    IF fbStateTimer.Q THEN
      fbStateTimer(IN:=FALSE);
      _nStarts := _nStarts + 1;
      IF bScriptAlive THEN
        nState := cStateRunning;    // is already running
      ELSE  
        RunPythonScript();          // start script
        nState := cStartScript;
			END_IF
		END_IF
  
  //Start Python script and wait until it starts
  cStartScript    :
    fbStateTimer(IN:=TRUE);
    _bBusy := TRUE;

    IF NOT fBScriptLauncher.bBusy AND bScriptAlive THEN 
      IF fBScriptLauncher.bError THEN //Launch error
        LogError(F_Concat2('Script start error=', TO_STRING(fBScriptLauncher.nErrId)));
        nState := cStateError;
      ELSE //Launch done and heartbeat ok
        nState := cStateRunning;
        fbStateTimer(IN:=FALSE);
			END_IF
    ELSIF fbStateTimer.Q THEN //Timeout error (could not start)
      IF fBScriptLauncher.bError THEN //Launch error
        ///LogError(F_Concat2('Script start error=', TO_STRING(fBScriptLauncher.nErrId)));
        LogError(F_Concat2('Script start error=', F_GetAdsErrStr(fBScriptLauncher.nErrId)));
      ELSE
        LogError('Script start error');
      END_IF
      nState := cStateError;
		END_IF
 
  //Script running with correct watchdog feedback
  cStateRunning   : 
    fbStateTimer(IN:=_bJobStartRequest);
    _bBusy := _bJobStartRequest;
    _bJobStopRequest := FALSE;
    _nStarts := 0;
    
    IF _bJobStartRequest AND bPythonNewJobDone THEN
      _bJobStartRequest:=FALSE;
      bPythonNewJobDone := FALSE; 
      fbStateTimer(IN:=FALSE);  
      nState := cStateJobActive;
    ELSIF NOT bScriptAlive THEN //Watchdog error
      LogError('Script watchdog error');
      nState := cStateError;
    ELSIF fbStateTimer.Q THEN //Job timeout error
      LogError('Script new job done error');
      nState := cStateError;
    ELSIF NOT bEnable THEN
      nState := cStateStop;
		END_IF
  
  //JobStarted
  cStateJobActive :
    fbStateTimer(IN:=_bJobStopRequest);
    _bBusy := _bJobStopRequest;
    
    IF _bJobStopRequest THEN
      nPythonNewJob := 0;
    END_IF;  
    
    IF _bJobStopRequest THEN
      _bJobStopRequest:=FALSE;
      fbStateTimer(IN:=FALSE);  
      nState := cStateRunning;
    ELSIF NOT bScriptAlive THEN //Watchdog error
      LogError('Script watchdog error');
      nState := cStateError;
    ELSIF fbStateTimer.Q THEN //Job timeout error
      LogError('Script new job done error');
      nState := cStateError;
    ELSIF NOT bEnable THEN
      nState := cStateStop;
		END_IF
  
  //Error  
  cStateError     :
    fbStateTimer(IN:=FALSE);  
    _bJobStartRequest:=FALSE;
    _bJobStopRequest:=FALSE;
    // reset error 
    IF _bResetError THEN
      _nStarts := 0;          // exit error 
      _nErrCtr := _nErrCtr + 1;
      nState := cStateStop ;
    ELSIF NOT bEnable THEN
      nState := cStateStop ;  // just stop
    ELSIF (_bKeepAlive AND _nStarts <= cMaxStartAttempts)  THEN
      _nErrCtr := _nErrCtr + 1;   // retry 
      nState := cStateStop ;
		END_IF
    
  //Stop 
  cStateStop  :
    StopPythonScript();
    nState := cStateStopping;

  // Stopping
  cStateStopping  :
    IF NOT fBScriptLauncher.bBusy THEN 
      IF fBScriptLauncher.bError THEN //Launch error
        LogError(F_Concat2('Script stop errror:', TO_STRING(fBScriptLauncher.nErrId)));
			END_IF
      nState := cStateIdle;
    END_IF

END_CASE
END_ACTION

METHOD JobStart
VAR_INPUT
  aJobName       : T_MaxString;
  aJobGuid       : T_MaxString;
  nJobImageWidth : UDINT;
  nJobImageHeigth  : UDINT;
  nCamFrameWidth : UDINT;
  pGridSettings  : POINTER TO ST_DefGridSettings;
END_VAR
_bJobStartRequest := TRUE;
_nJobIdCtr := _nJobIdCtr + 1;
nPythonNewJob := _nJobIdCtr;

aPythonJobName := aJobName;
aPythonJobGuid := aJobGuid;
nPythonImageWidth := nJobImageWidth * GVL_Deformation.nC_GridSubReso;
nPythonImageHeight :=nJobImageHeigth * GVL_Deformation.nC_GridSubReso;
nPythonCamFrameWidth := nCamFrameWidth * GVL_Deformation.nC_GridSubReso;
IF pGridSettings <> 0 THEN
  nPythonImageOffsetY := pGridSettings^.nGridImageOffsetY * GVL_Deformation.nC_GridSubReso;
  nPythonGridPitchX := pGridSettings^.nGridPitchX * GVL_Deformation.nC_GridSubReso;
  nPythonGridPitchY := pGridSettings^.nGridPitchY * GVL_Deformation.nC_GridSubReso;
  nPythonGridSizeX := pGridSettings^.nGridSizeX * GVL_Deformation.nC_GridSubReso;
  nPythonGridSizeY := pGridSettings^.nGridSizeY * GVL_Deformation.nC_GridSubReso; 
END_IF
END_METHOD

METHOD JobStop : BOOL
VAR_INPUT
END_VAR
_bJobStopRequest:=TRUE;
END_METHOD

{attribute 'monitoring':='call'}
PROPERTY nErrorId : UDINT
GET
nErrorId := _nErrId;
END_GET
END_PROPERTY

(*
  Register CT to script.
  :return: TRUE if success.
*)
METHOD RegisterCT : BOOL
VAR_INPUT
  nCTIdx  : UDINT;  // ct memory index
END_VAR
IF NOT bScriptAlive THEN RETURN; END_IF  // script not ready, ignore request

nContainerToRegister := UDINT_TO_DINT(nCTIdx);
RegisterCT := TRUE;
END_METHOD

METHOD RemoveCT : BOOL
VAR_INPUT
    nCTID : UDINT;
END_VAR
IF NOT bScriptAlive THEN RETURN; END_IF  // script not ready, ignore request

nContainerToDelete := UDINT_TO_DINT(nCTID);

RemoveCT := TRUE;
END_METHOD

METHOD PRIVATE RunPythonScript : BOOL
VAR_INPUT
END_VAR
VAR
  ams_host : STRING;
  ams_port : UINT;
  cmd : STRING;
END_VAR
// config launcher cmd line for script
//   e.g. fBScriptLauncher.Start('172.17.7.143.1.1 851 PRG_PRINT.fbWorkerDefGrid_Python.fbPythonInterface --sim_mode');

// get parameter dynamically
ams_host := PRG_SYSTEMBASE.sO_AmsNetIdLocalHost;  // localhost
ams_port := TwinCAT_SystemInfoVarList._AppInfo.AdsPort;
cmd := F_Concat5(ams_host,' ',TO_STRING(ams_port),' ',sPythonInterfacePath);
fBScriptLauncher.sStartScriptName := 'start.bat';
fBScriptLauncher.sStopScriptName  := 'stop.bat';
fBScriptLauncher.Start(cmd);
END_METHOD

METHOD PRIVATE StopPythonScript
VAR_INPUT
END_VAR
fBScriptLauncher.Stop(nPID := THIS^.nPythonPID);
END_METHOD

{attribute 'monitoring':='call'}
PROPERTY tWatchdogTime : TIME
GET
tWatchdogTime := fbWatchdog.ET;
END_GET
END_PROPERTY

END_FUNCTION_BLOCK

// ---- POUs/Print/DefGrid/FB_StartPositionDummy.TcPOU
(*
  A start position detection function block dummy.
  A dummy implementation to simulate start triggers at desired positions.
*)
FUNCTION_BLOCK FB_StartPositionDummy EXTENDS FB_BasePrint IMPLEMENTS I_StartPosDetect, I_PrintStatusClient, I_Sim
VAR_INPUT
  bTrigger                    : BOOL;       // manual trigger
  lPosition                   : DINT;       // current position [SubPx]
  fSpeed                      : LREAL;      // current speed [m/s]
  fResolution                 : LREAL;      // current print resolution [dpi*SubPx]
END_VAR

VAR
  // properties
  _bSim               : BOOL;       // simulatio mode active (PROPERTY)
  _bCreateTrigger     : BOOL;       // create new CT trigger (PROPERTY)
  _nStartPosX0        : DINT;       // create position for CT (absolut) [SubPx] (PROPERTY)
  _bAutoTrigger       : BOOL;       // automatic sheet triggers
  
  // config
  iJobDefinition      : CalmarCompPrint.I_JobDefinition;
  
  // local helper
  rfNewCT             : RF_TRIG;    // trigger new ct
  nSheetLength        : DINT;       // sheet length in [SubPx]
  nSheetGap           : DINT;       // sheet gap in [SubPx]
  nSheetEndPosition   : DINT;       // sheet end position [SubPx]
  nNextSheetPosition  : DINT;       // next trigger location
  fSheetPerHour       : LREAL;      // sheets per hour
  fSheetSpeed         : LREAL;      // [m/min] speed meter per minute
  tCheckTrigger       : TON;
  
  tCurrentTimeStamp   : T_DCTIME64; // get current timestamp
  fCurrentTimeStamp   : LREAL;      // current timestamp
  fSensorTimeStamp    : LREAL;      // sensor timestamp
  fDeltaDistance      : LREAL;      // distance that the substrate moved between the detection and the treatment of the information [m]
  
  rfTrig_Sim          : RF_TRIG;
END_VAR

VAR PERSISTENT
  // simulation configuration
  fSheetLength   : LREAL := 0.5;    // [m] sheet length (local or per job given)
  fSheetGap      : LREAL := 0.12;   // [m] gap between two sheets
END_VAR

// checks and fixes
IF iJobDefinition = 0 THEN RETURN; END_IF
IF fSpeed = 0 THEN RETURN; END_IF
IF fSheetLength = 0 THEN fSheetLength := 1; END_IF
IF fResolution = 0 THEN fResolution := 600*32; END_IF
rfTrig_Sim(CLK:=_bSim);
IF    rfTrig_Sim.RT THEN SimEnter(); 
ELSIF rfTrig_Sim.FT THEN SimExit(); END_IF

IF NOT _bSim THEN RETURN; END_IF

// calculations
fSheetSpeed := fSpeed * 60;  // [m/s] -> [m/min]
nSheetGap := F_MeterToSubPixel(fPosMeter := fSheetGap, fResoSubPx := fResolution);  // [m] -> [SubPx]
fSheetPerHour := (60*60)/((fSheetLength+fSheetGap)/fSpeed);
nSheetLength := F_MeterToSubPixel(fPosMeter := fSheetLength, fResoSubPx := fResolution);  // [mm] -> [SubPx]
nNextSheetPosition := _nStartPosX0 + nSheetLength + nSheetGap; 
tCheckTrigger(PT:=TO_TIME(((fSheetLength+fSheetGap)/fSpeed)*1000));

// internal trigger creation
IF (lPosition - nNextSheetPosition) > 0 AND _bAutoTrigger THEN
  bTrigger := TRUE;
  tCheckTrigger(IN:=FALSE);
  tCheckTrigger(IN:=TRUE);
END_IF

// on trigger
rfNewCT(CLK := bTrigger, RT => _bCreateTrigger);
IF _bCreateTrigger THEN   // new ct created
  bTrigger := FALSE;  // reset trigger
  
  (* Calculate the current and sensor time stamp (keep old code not really necessary because we use current timestamp)*)
  tCurrentTimeStamp := F_GetCurDcTaskTime64();
  fCurrentTimeStamp := (ULINT_TO_LREAL(tCurrentTimeStamp )) / 1_000_000.0; (*in ms*)
  fSensorTimeStamp  := fCurrentTimeStamp;
  fDeltaDistance := (fCurrentTimeStamp - fSensorTimeStamp) * 0.001 * fSpeed;  (*Distance that the substrate moved between the detection and the treatment of the information [m]*)
  
  // sheet start and sheet end pos in [SubPx]
  _nStartPosX0     := lPosition - F_MeterToSubPixel(fPosMeter := fDeltaDistance, fResoSubPx := fResolution);
  nSheetEndPosition := _nStartPosX0 + nSheetLength;
END_IF

{attribute 'monitoring' := 'call'}
(*Simulation is enabled set/get*)
PROPERTY bSimEnable : BOOL
GET
bSimEnable := _bSim;
END_GET
SET
_bSim := bSimEnable;
END_SET
END_PROPERTY

(*
  A new container detected.
  NOTE: a pulse only
*)
PROPERTY bStartTrig : BOOL
GET
bStartTrig := _bCreateTrigger;
END_GET
END_PROPERTY

(*
  A valid container detected.
*)
PROPERTY bValid : BOOL
GET
bValid := TRUE;
END_GET
END_PROPERTY

METHOD mJobPause
END_METHOD

METHOD mJobStart
VAR_INPUT
	sJobDef	: CalmarCompPrint.I_JobDefinition;
END_VAR
IF sJobDef = 0 THEN LogError('JobStart: no sJobDef given'); RETURN; END_IF

iJobDefinition := sJobDef;    // current job definition
fSheetLength := iJobDefinition.fSubstrateDepth;
END_METHOD

METHOD mJobStop
VAR_INPUT
	sStatus	: CalmarCompPrint.I_JobStatus;
END_VAR
iJobDefinition := 0;    // delete job definition
END_METHOD

METHOD mProduced
VAR_INPUT
	(* current progress*)
	sProgress	: CalmarCompPrint.I_JobProgress;
END_VAR
; // nothing to do
END_METHOD

(*
  Detected start position X0 (absolute) in [SubPx].
*)
PROPERTY nStartPositionX0 : DINT
GET
nStartPositionX0 := _nStartPosX0;
END_GET
END_PROPERTY

METHOD SimEnter : BOOL
LogInfo('Enter start position creator simulation');
_bSim := TRUE;

_nStartPosX0 := lPosition;
nSheetEndPosition := lPosition;
nNextSheetPosition := lPosition;
END_METHOD

METHOD SimExit : BOOL
LogInfo('Exit start position creator simulation');
_bSim := FALSE;
END_METHOD

END_FUNCTION_BLOCK

// ---- POUs/Print/DefGrid/FB_WorkerDefGrid_Delete.TcPOU
FUNCTION_BLOCK FB_WorkerDefGrid_Delete EXTENDS FB_WorkerDefGrid

METHOD PROTECTED  Attach : BOOL
VAR_INPUT
  iCT              : I_CT;                         (*container at triggered event position*)
END_VAR
IF SUPER^.Attach(iCT:=iCT) THEN

  // directyl release & delete the CT 
  Release(iCT:=_pAttachedCt^);

END_IF
END_METHOD

METHOD   mJobStart
VAR_INPUT
	sJobDef	: CalmarCompPrint.I_JobDefinition;
END_VAR
END_METHOD

METHOD  mJobStop
VAR_INPUT
	sStatus	: CalmarCompPrint.I_JobStatus;
END_VAR
END_METHOD

METHOD Release : BOOL
VAR_INPUT
  iCT              : I_CT;                         (*container at triggered event position*)
END_VAR
IF SUPER^.Release(iCT := iCT) THEN
  
  // it's the last worker so distroy attached CT
  IF _pCTM <> 0 THEN
    LogLvl(Lvl:=E_LogSeverity.Debug, Msg:=F_Concat2('DestroyCT: ', TO_STRING(iCT.pCT^.iId)));
    _pCTM^.DestroyCT(iCT:=iCT);
  END_IF
  
END_IF
END_METHOD

METHOD  work
SUPER^.work();

// release should already be done in attach
IF _pAttachedCt <> 0 THEN
  Release(iCT:=_pAttachedCt^);
END_IF
END_METHOD

END_FUNCTION_BLOCK

// ---- POUs/Print/DefGrid/FB_WorkerDefGrid_Print.TcPOU
FUNCTION_BLOCK FB_WorkerDefGrid_Print EXTENDS FB_WorkerDefGrid IMPLEMENTS I_PrintSubsystem
VAR_INPUT
  nEncoderPos           : DINT;   // Absolute virtual encoder
  bHardwareSync         : BOOL;
  bHardwareHold         : BOOL;
  {warning 'TODO: refactor according WorkerPrintWEU offsets in [m] and worker position without DetectToPrintDist?'}
  fPrintStartOffset     : LREAL;  // Offset from Module reference (configurative PU/PM/PG/PA ADS offset)
  fDetectOffset         : LREAL;  // StartDetect to Modoule reference
  fPrintYOffset         : LREAL;  // Y-Shift in ram memory
  fMasterSpeed          : LREAL;  // Speed [m/s]
  fPUElevation          : LREAL;  // PU distance from substrate [m]
  fPUPlate1_Temperature : LREAL;  // PU Plate1 temperature
  fPUPlate2_Temperature : LREAL;  // PU Plate2 temperature
END_VAR

VAR_OUTPUT
  bPrintActive          : BOOL;   // A print is activated / started
END_VAR

VAR
  // print
  // - references
  _pAdsPg            : POINTER TO FB_ADS_PG;      // pg ads reference (for pa)

  // grid specific
  // - references
  _iParamMediator    : I_ParamMediator;
    
  sDefGridSettings   : ST_DefGridSettings;  
  fCurrentColumnPos  : LREAL; // Currently column position
  fCurrentPreCharge  : LREAL; // Currently to be precharged
  nChargedColumns    : UDINT; // Already charged columns

  fbDropSpeedComp    : FB_DropSpeedComp;  
  bShowDropSpeedSetup: BOOL;

  fbPs               : FB_PS;
  fbPa               : FB_PA;
  fB_PcAdapter       : FB_PC_Adapter;

  _fPrintStartOffset : LREAL;   // internal print start offset (distance Cam -> PG1 + PG Offset + PU offset)
  _fWorkerOffset     : LREAL;   // worker offset from X0 static
  _nPosX0            : DINT;    // X0 for last attached CT (detected postion)
  _nPosXS            : DINT;    // XS for last attached CT (shifted print start position)
  _nPosXDelta        : DINT;    // Shift value X0 -> XS
  _fPosY             : LREAL;   // Y shift for last attached CT
  _fCurrentImgDepth  : LREAL;   // Job: current image length [m]
  _nPosDeltaToPrint  : DINT;    // delta pos in [SbuPx] from attach to print
  _bPaStarted        : BOOL;
  _bPaStartRequested : BOOL;
  fBStartTimeout     : TON;
  rTrigSync          : R_TRIG;
  _bForceDefGridOff  : BOOL;    // force deformation grid stream to ph off (send 0)
  _fPrintUnitWidth   : LREAL;   // print unit width [m]
  // grid settings
  _iPhGrid           : I_Correction_Grid;
  _sPhGridHwCfg      : ST_GridHwCfg;
    
  (*grid limit*)
  _fLimitCorrectionX : LREAL;     // correction limit in y (abs) [px]
  _fLimitCorrectionY : LREAL;     // correction limit in y (abs) [px]
  _bGridWasLimited   : BOOL;      // streamed grid was limited
    
  (*Messaging*)
  _bMsgInitialized   : BOOL;
  fb_MsgQueue        : FB_MSG_QUEUE;                        (*Message queue*)
  fb_MsgHandler      : FB_MSG_HANDLER;                      (*Message handler*)
  sL_MsgConfig       : ST_MSG_CONFIG;                       (*Message config*)
  fb_Msg             : ARRAY [1..iC_NUM_MSG] OF FB_MESSAGE; (*Messages*)
END_VAR

VAR PERSISTENT
  _fColumnsToPrecharge : LREAL := nC_COLUMNS_TO_PRECHARGE;
  _fStartShiftOffset   : LREAL := fC_START_SHIFT_OFFSET;
  _fStartShiftFactor   : LREAL := fC_START_SHIFT_FACTOR;
END_VAR

VAR CONSTANT
  iC_NUM_MSG               : UDINT := 5;
  nC_COLUMNS_TO_PRECHARGE  : LREAL := 2.1;
  fC_GRIDPOINT_STREAM_TIME : LREAL := 0.0025;     // time to stream one point [s]
  fC_START_SHIFT_FACTOR    : LREAL := -0.031;
  fC_START_SHIFT_OFFSET    : LREAL := -0.01;
END_VAR

IF NOT bInitialized THEN RETURN; END_IF

//TODO Add error/warnings
bError := FALSE;
nError := 0;

fbDropSpeedComp(fMasterSpeed:=fMasterSpeed, fDropTravelDistance:=fPUElevation);

//Start offset update
IF _fPrintStartOffset <> (fPrintStartOffset) THEN //Worker position changed
  IF _pAttachedCt = 0 THEN //Update only without attached container
    _fPrintStartOffset :=fPrintStartOffset;
	END_IF
END_IF

//Worker position update
IF _fWorkerPosition <> (_fPrintStartOffset + (_fStartShiftOffset + _fStartShiftFactor * fMasterSpeed)) THEN //Worker position changed (camera settings change)
  setupPosition();
END_IF

(*---- Messaging -----------------------*)
IF _bMsgInitialized THEN
  fb_MsgHandler();
  //fB_Msg[1](bI_Status := dfsdfdsf);
  fb_MsgQueue();
END_IF

PROPERTY aPaState : STRING
GET
aPaState := fbPa.aPaState;
END_GET
END_PROPERTY

METHOD PROTECTED  Attach : BOOL
VAR_INPUT
  iCT              : I_CT;                         (*container at triggered event position*)
END_VAR
Attach:=FALSE;

IF SUPER^.Attach(iCT:=iCT) THEN
  // Additional worker checks
    // - job is valid?
  IF _pAttachedCt^.pJob = 0 OR NOT _bJobActive THEN
    Release(iCT:=iCT);
    RETURN;   // do not print
  
  // CT valid & CT present
  ELSIF NOT _pAttachedCt^.bValid OR NOT _pAttachedCt^.bProductPresent THEN
    Release(iCT:=iCT);
    RETURN;   // do not print
  
  // Ignore start due to hardware hold  
  ELSIF bHardwareHold THEN
    _pNewAttached^.AbortDeformation(sReason:=EC_Print.ecPaAbortHold.Desc, Src:=_pEcSrc^, bHideLog:=TRUE);
    Release(iCT:=iCT);
    RETURN;   // do not print
  
  // - OK attach
  ELSE
    Attach := TRUE;
	END_IF
  
  
  //Prepare print station
  sDefGridSettings := _pAttachedCt^.sDefGridSettings;
  // fix some potential errors
  IF sDefGridSettings.nGridPitchX = 0 THEN sDefGridSettings.nGridPitchX :=1024; LogError(F_concat2('grid not configured, set default nGridPitchX=',TO_STRING(sDefGridSettings.nGridPitchX))); END_IF
  IF sDefGridSettings.nGridPitchY = 0 THEN sDefGridSettings.nGridPitchY :=1024; LogError(F_concat2('grid not configured, set default nGridPitchY=',TO_STRING(sDefGridSettings.nGridPitchY))); END_IF
  
  fbPs.bPrintEnable := iCT.bValid AND iCT.bProductPresent;
  fbPs.setGrid(sGrid:=sDefGridSettings);
  nChargedColumns := 0;

  //Start print, PA should be in READY or DONE
  
  // Set X print position
  _nPosX0 :=    _pAttachedCt^.nPosPrint_X0   {warning 'TODO: please write this in DMAX CreateCT CTM'}
              //- General Shift
              - F_MeterToSubPixel(fbDropSpeedComp.fDropPlacementError, _fPrintResolution*_fSubPxResolution); // - drop compensation*)
  _nPosXDelta := F_MeterToSubPixel(_fPrintStartOffset, _fPrintResolution*_fSubPxResolution); // + PG/PA Shift (additional PG offset 0 for firstLine)
  
  _nPosXS := _nPosX0 + _nPosXDelta;
  fB_PcAdapter.setPrintStartPos(nX0:=_nPosXS);
  
  // Set Y print position
  _fPosY := fPrintYOffset;
  fB_PcAdapter.setPrintYShift(nYShift:=FC_LREAL_TO_DINT(_fPosY));

  // check
  IF _nPosXS < nEncoderPos THEN
    LogWarning(Msg:=F_Concat4('Print start position:', TO_STRING(_nPosXS) ,' < Encoder position:', TO_STRING(nEncoderPos)));
	END_IF
  
  // save current distance to print position
  _nPosDeltaToPrint := _nPosXS - _iCTTracker.getPosAbs();   {warning 'TODO: to test if this matches after the change'}
  checkGridTiming();
  
  IF fbPa.printStart() THEN
    _bPaStarted := FALSE;
    _bPaStartRequested := TRUE;
    Attach:=TRUE;
    LogLvl(Lvl:=E_LogSeverity.Debug, F_Concat2('printStart:', _pAttachedCt^.print(0)));  // print container
    LogLvl(Lvl:=E_LogSeverity.Debug, F_Concat4('> XS:', TO_STRING(_nPosXS), ' = X0:', TO_STRING(_nPosX0)));
    LogLvl(Lvl:=E_LogSeverity.Debug, F_Concat4( 
                                         ' + shStartOffs:', TO_STRING(F_MeterToSubPixel(_fPrintStartOffset,_fPrintResolution*_fSubPxResolution)),
                                         ' - shDropComp:', TO_STRING(F_MeterToSubPixel(fbDropSpeedComp.fDropPlacementError,_fPrintResolution*_fSubPxResolution))
                                         ));
  ELSE  
    LogError(Msg:='PA not ready to start at attach');
    Release(iCT := iCT);
	END_IF
  
ELSE
  // parent attach failed case
END_IF
END_METHOD

PROPERTY bJobActive : BOOL
GET
bJobActive := _bJobActive;
END_GET
END_PROPERTY

PROPERTY bPausePrintCanEx : BOOL
GET
bPausePrintCanEx := FALSE; //Not implemented
END_GET
END_PROPERTY

PROPERTY bPcEnabled : BOOL
GET
bPcEnabled := fB_PcAdapter.bPcEnable;
END_GET
END_PROPERTY

PROPERTY bPrintEnabled : BOOL
GET
bPrintEnabled := _bEnable;
END_GET
END_PROPERTY

PROPERTY bPrinting : BOOL
GET
bPrinting := fbPa.bPrinting;
END_GET
END_PROPERTY

PROPERTY bPrintReady : BOOL
GET
bPrintReady := fbPa.bReady;
END_GET
END_PROPERTY

PROPERTY bQueueEmpty : BOOL
GET
bQueueEmpty := NOT fB_PcAdapter.bJobValid;
END_GET
END_PROPERTY

PROPERTY bStartPrintCanEx : BOOL
GET
bStartPrintCanEx := fbPa.bStartCanEx;
END_GET
END_PROPERTY

PROPERTY bStopPrintCanEx : BOOL
GET
bStopPrintCanEx := fbPa.bStopCanEx;
END_GET
END_PROPERTY

METHOD PRIVATE checkGridTiming : BOOL
VAR
END_VAR
// check for timing problems
IF fMasterSpeed <> 0 THEN

  // - check pre-charge at beginning
  IF _fColumnsToPrecharge * fC_GRIDPOINT_STREAM_TIME * _sPhGridHwCfg.nGridRoiRows >= F_SubPixelToMeter(lPosSubPx:=_nPosDeltaToPrint, fResSubPx:=_fPrintResolution*_fSubPxResolution) / fMasterSpeed  THEN
    LogError('Machine too fast for grid stream (for pre-charge at attach)');
  END_IF
  
 // - check charge time needed per columns vs machine speed and grid-sizeY
 IF fC_GRIDPOINT_STREAM_TIME * _sPhGridHwCfg.nGridRoiRows >= F_SubPixelToMeter(lPosSubPx:=TO_DINT(sDefGridSettings.nGridPitchX), fResSubPx:=_fPrintResolution) / fMasterSpeed THEN
   LogError('Machine too fast for grid stream (time rows per column)');
 END_IF

END_IF
END_METHOD

(*
  Limit correction to boundaries
  :return: TRUE if limited
*)
METHOD PRIVATE correctionLimit : BOOL
VAR_INPUT
  pPoint : POINTER TO ST_DeformationPointAccurate;
END_VAR
VAR
  bLimited : BOOL;
  nExeedX, nExeedY : LREAL;
END_VAR
// limit point correction to boundaries and inform
IF    pPoint^.dx >= _fLimitCorrectionX    THEN nExeedX := pPoint^.dx; pPoint^.dx := _fLimitCorrectionX;    bLimited:=TRUE; 
ELSIF pPoint^.dx <= -1*_fLimitCorrectionX THEN nExeedX := pPoint^.dx; pPoint^.dx := -1*_fLimitCorrectionX; bLimited:=TRUE;
ELSIF pPoint^.dy >= _fLimitCorrectionY    THEN nExeedY := pPoint^.dy; pPoint^.dy := _fLimitCorrectionY;    bLimited:=TRUE;
ELSIF pPoint^.dy <= -1*_fLimitCorrectionY THEN nExeedY := pPoint^.dy; pPoint^.dy := -1*_fLimitCorrectionY; bLimited:=TRUE;
END_IF
IF bLimited THEN 
  LogLvl(Lvl:=E_LogSeverity.Warning, Msg:=F_Concat5( 'Point=',TO_STRING(pPoint^.index),
                                                     F_Concat5(' c:r(',TO_STRING(pPoint^.col),'/',TO_STRING(pPoint^.row), ') '),
                                                     F_Concat4('dx:', TO_STRING(nExeedX), ' dy:', TO_STRING(nExeedY)),
                                                     ' correction exceeded limit')); 
END_IF

_bGridWasLimited := SEL(bLimited, FALSE, TRUE);
correctionLimit := bLimited;
END_METHOD

// current job image length in [m]
PROPERTY fImageLength : LREAL
GET
fImageLength := _fCurrentImgDepth;
END_GET
END_PROPERTY

PROPERTY fMaxPrintSpeed : LREAL
GET
fMaxPrintSpeed := 0;  // TODO: when i_pc_adapter has the info from pc/ph
END_GET
END_PROPERTY

(*
  Max. supported speed [m/s], 0 if not available
*)
{attribute 'monitoring':='call'}
PROPERTY fMaxSpeed : LREAL
GET
VAR
  nSpeedMpMin : DINT;
END_VAR
nSpeedMpMin := SEL(bWorkerEnable AND _pAdsPg <> 0, 0, _pAdsPg^.lMaxPrintSpeed);
fMaxSpeed := TO_LREAL(nSpeedMpMin)/60;
END_GET
END_PROPERTY

{attribute 'monitoring':='call'}
PROPERTY fStartShiftFactor : LREAL
GET
fStartShiftFactor := _fStartShiftFactor;
END_GET
SET
_fStartShiftFactor := fStartShiftFactor;
END_SET
END_PROPERTY

{attribute 'monitoring':='call'}
PROPERTY fStartShiftOffset : LREAL
GET
fStartShiftOffset := _fStartShiftOffset;
END_GET
SET
_fStartShiftOffset := fStartShiftOffset;
END_SET
END_PROPERTY

METHOD PROTECTED gridUpdate : BOOL
VAR_INPUT
  bEnableDeformation : BOOL;      // enable correction update, else correction (0/0) is written
  fPosRelToAttach : LREAL;        // position relative to attach of this worker
END_VAR
VAR
  sPoint : ST_DeformationPointAccurate;
  nRow : UDINT;
  bWasSet : BOOL;
  nAvailPoints : UDINT;
  nConvErr : UDINT;
END_VAR
VAR_INST
  nAvailPoints_mem : UDINT;
END_VAR
//TODO: rewrite this method to look cleaner (less if else)
gridUpdate:=TRUE;

// calculate grid column position
IF sDefGridSettings.nGridPitchX <> 0 THEN
  fCurrentColumnPos := fPosRelToAttach / (sDefGridSettings.nGridPitchX * _fSubPxResolution);   // calc grid column position relative to worker
END_IF

//Check for next correction update 
IF fCurrentColumnPos + _fColumnsToPrecharge > nChargedColumns AND nChargedColumns <= sDefGridSettings.nGridSizeX THEN
  IF bEnableDeformation THEN 
    // sync deformation points
    {warning 'TODO FIX: WHILE'}
    fCurrentPreCharge := fCurrentColumnPos + _fColumnsToPrecharge;
    WHILE FLOOR(fCurrentPreCharge) > nChargedColumns AND nChargedColumns <= sDefGridSettings.nGridSizeX DO
      nAvailPoints := _pAttachedCt^.nAvailableGridPoints;
      IF nAvailPoints >= sDefGridSettings.nGridSizeY * (nChargedColumns+1) THEN // Complete column available?
        nAvailPoints_mem := 0;
        LogLvl(Lvl:=E_LogSeverity.Debug, Msg:=F_Concat2('Charge CG col: ',TO_STRING(nChargedColumns)));
        FOR nRow := 0 TO sDefGridSettings.nGridSizeY - 1 DO
          // get points
          IF _pAttachedCt^.getDeformationPoint(nCol:=nChargedColumns, nRow:=nRow, nSel:=0, sPoint=>sPoint, bWasSet=>bWasSet) THEN
          
            IF NOT bWasSet THEN LogWarning(F_Concat5('Point[c(',TO_STRING(nChargedColumns),')/r(', TO_STRING(nRow),')] was not set')); END_IF  
                      
            // correction limitation
            correctionLimit(pPoint:=ADR(sPoint));
            
            // send point
            IF NOT fbPs.newGridPoint(sPoint:=sPoint) THEN
               LogError(Msg:='stream new point failed');
               gridUpdate:=FALSE;
               RETURN;
            END_IF
          ELSE
            LogError(Msg:='get new grid point failed');
            gridUpdate:=FALSE;
          END_IF
        END_FOR
        
        nChargedColumns := nChargedColumns + 1;
      ELSE
        IF nAvailPoints > nAvailPoints_mem THEN // log once or after every update of new available poinst
          LogError(Msg:='point column expected but not available');
        END_IF
        nAvailPoints_mem := nAvailPoints;
        gridUpdate:=FALSE;
        RETURN;
      END_IF 
    END_WHILE
  ELSE
    // send points with no deformation
      FOR nRow := 0 TO sDefGridSettings.nGridSizeY - 1 DO
        MEMSET(destAddr:=ADR(sPoint), fillByte:=0, n:=SIZEOF(sPoint));
        sPoint.col := TO_DINT(nChargedColumns);
        sPoint.row := TO_DINT(nRow);
        IF NOT fbPs.newGridPoint(sPoint:=sPoint) THEN
           LogError(Msg:='stream new point failed');
           gridUpdate:=FALSE;
           RETURN;
        END_IF
    END_FOR
    nChargedColumns := nChargedColumns + 1;
	END_IF
END_IF
END_METHOD

METHOD InitMsg : BOOL
VAR_INPUT
  pMsgInterface : POINTER TO ST_ADS_MSG_IF;
END_VAR
VAR
  nCtr : UDINT;
END_VAR
IF pMsgInterface = 0 THEN RETURN; END_IF

(*Messaging*)
sL_MsgConfig.bI_Enable       := TRUE;
sL_MsgConfig.pI_FbMsgHandler := ADR(fb_MsgHandler);
fb_MsgHandler.pI_MsgQueue    := ADR(fb_MsgQueue);
fb_MsgQueue.pI_MsgInterface  := pMsgInterface;
fb_MsgQueue.cI_MaxElement    := 6;

(*Messages*)
FOR nCtr := 1 TO iC_NUM_MSG DO
  fb_Msg[nCtr].pI_MsgConfig       := ADR(sL_MsgConfig);
  fb_Msg[nCtr].iI_MsgLocation     := 0;
END_FOR
//fb_Msg[1].iI_MsgNumber       := ;
// ...

_bMsgInitialized := TRUE;
END_METHOD

METHOD InitWorkerPrint : BOOL
VAR_INPUT
  pAdsPg                : POINTER TO FB_ADS_PG;       // pg ads reference (worker prints ads)
  iDefGridParamMediator : I_ParamMediator;
  fPrintUnitWidth       : LREAL;     // print unit width [m]
  fLimitCorrectionX     : LREAL;     // correction limit in y (abs) [px]
  fLimitCorrectionY     : LREAL;     // correction limit in y (abs) [px]
END_VAR
IF NOT bInitialized THEN LogError('Base Worker not initialized! call init() before'); RETURN; END_IF
IF pAdspg = 0 THEN LogError('InitWorkerPrint: invalid parameter proviced'); RETURN; END_IF
IF iDefGridParamMediator = 0 THEN bInitialized := FALSE; LogError('Invalid parameter, no valid param mediator'); RETURN; END_IF

// worker specific init
_pAdsPg := pAdsPg;
_iParamMediator := iDefGridParamMediator;

//Print Aggregate
_fPrintUnitWidth   := fPrintUnitWidth;
_fLimitCorrectionX := ABS(fLimitCorrectionX);
_fLimitCorrectionY := ABS(fLimitCorrectionY);

fbPa.bSyncAfterDone := FALSE;
fbPa.init(iPcAdapter := fB_PcAdapter, iPsInterface := fbPs);
END_METHOD

METHOD   mJobStart
VAR_INPUT
	sJobDef	: CalmarCompPrint.I_JobDefinition;
END_VAR
// Config workers static variables
_fCtSecurityReleasePos := F_MeterToSubPixel(fPosMeter:=(1.5 *sJobDef.fImageDepth) /1000, fResoSubPx:=_fPrintResolution*_fSubPxResolution);

IF NOT bWorkerEnable THEN RETURN; END_IF  // only if enabled

fbPa.jobStart(bEndless:=sJobDef.isEndless());

_bJobActive := TRUE;
_fCurrentImgDepth := sJobDef.fImageDepth/1000;

// grid settings update
IF _iPhGrid <> 0 THEN _sPhGridHwCfg := _iPhGrid.getGridHwCfg(); END_IF
END_METHOD

METHOD  mJobStop
VAR_INPUT
	sStatus	: CalmarCompPrint.I_JobStatus;
END_VAR
fbPa.jobStop();
_bJobActive := FALSE;
END_METHOD

PROPERTY pMsgConfig : POINTER TO ST_MSG_CONFIG
GET
pMsgConfig := ADR(sL_MsgConfig);
END_GET
END_PROPERTY

METHOD registerPc : BOOL
VAR_INPUT
  iNewPC : I_PC;
END_VAR
registerPc := fB_PcAdapter.registerPc(iNewPC := iNewPC);
END_METHOD

METHOD registerPh : BOOL
VAR_INPUT
  iPH : I_PH;
END_VAR
//Attach head to print station
IF iPH <> 0 THEN
  fbPs.registerPh(iNewPh:=iPH);
  _iPhGrid := iPH.iGridCorrection;
END_IF
END_METHOD

METHOD setupPosition
IF _pAttachedCt <> 0 THEN RETURN; END_IF    // Update only without attached container

// WorkerPosition =  PU<-CAM + CAM<-SheetDetect + StartShift calculated (with speed)
fPosition := _fPrintStartOffset + (_fStartShiftOffset + _fStartShiftFactor * fMasterSpeed);
END_METHOD

PROPERTY sPcFlags : CalmarCompPrint.ST_PC_FLAGS
GET
sPcFlags := fB_PcAdapter.sPcFlags;
END_GET
END_PROPERTY

PROPERTY sPcState :  CalmarCompPrint.ST_PG_STATUS
GET
VAR
  sJobStatus : ST_JobProgress;
END_VAR
sPcState.bStartPrintCanEx := fBPa.bStartCanEx;
sPcState.bStartPrintExec  := fBPa.bStartExec;
sPcState.bStopPrintCanEx  := fBPa.bStopCanEx;
sPcState.bStopPrintExec   := fBPa.bStopExec;
sPcState.bPausePrintCanEx := FALSE;       // obsolete ???
sPcState.bPausePrintExec  := FALSE;       // obsolete ???
sPcState.bReady           := fB_PcAdapter.bAllReady OR fB_PcAdapter.bAllDone;
sPcState.bError           := fB_PcAdapter.bError;
sPcState.bPrinting        := fB_PcAdapter.bAllPrinting;
sPcState.bLoad            := fB_PcAdapter.bAllPreparing;
sPcState.bArmed           := fB_PcAdapter.bAllPrinting OR fB_PcAdapter.bAllReady OR fB_PcAdapter.bAllDone OR fB_PcAdapter.bAllPreparing;
sPcState.bEnabled         := bWorkerEnable;
sPcState.bStartStrb       := fBPa.bStartStrb;
sPcState.bPcEnabled       := fB_PcAdapter.bPcEnable;
sPcState.lProductCount    := 0;            // obsolete ???
sPcState.sJobStatus       := sJobStatus;   // obsolete ???
END_GET
END_PROPERTY

METHOD  work
VAR
  bDeformErr : BOOL;
  nDeformStep : E_DeformationStep;
END_VAR
SUPER^.work();

(*Update virtual encoder on all controller boards*)
fB_PcAdapter.setEncoderPos(nEncoderPos);
fB_PcAdapter();

(*Call print aggregate*)
rTrigSync(CLK:=bHardwareSync); 
IF rTrigSync.Q THEN fbPa.sync(); END_IF   // external sync
fbPa.bHold := bHardwareHold;              // external hw hold
fbPa();

fBStartTimeout(IN := _bPaStartRequested,PT := T#60MS);

IF _pAttachedCt <> 0 AND bWorkerEnable THEN // Work only with attached container
  
  // check for generic error
  IF _pAttachedCt^.bValid AND bHardwareHold THEN
    // abort during printing
    _pNewAttached^.AbortDeformation(sReason:=EC_Print.ecPaAbortHold.Desc, Src:=_pEcSrc^, bHideLog:=TRUE);
  END_IF

  // Grid update
  bDeformErr := _pAttachedCt^.getDeformationStatus(eDStep=>nDeformStep);
  {warning 'TODO: re-enable gridUpdate()'}
(*
  IF NOT bDeformErr AND nDeformStep >= E_DeformationStep.gridStarted AND NOT _bForceDefGridOff THEN 
    IF NOT gridUpdate(bEnableDeformation:=TRUE) THEN
      _pAttachedCt^.AbortDeformation(sReason:='WorkerPrint: deformation point update failed', Src:=_pEcSrc^);
    END_IF
  ELSE
    // not started or error already --> erase deformation points
    gridUpdate(bEnableDeformation:=FALSE);
  END_IF  
*)  
  // PA control
  IF _bPaStartRequested THEN
    IF fbPa.bPrinting THEN
      _bPaStarted := TRUE;
      _bPaStartRequested := FALSE;
    ELSIF fBStartTimeout.Q THEN //Stop print at timeout to make ready for next container
      _bPaStarted := FALSE;
      _bPaStartRequested := FALSE;
      fbPa.printStop(bSyncedStop:=FALSE);
      _pNewAttached^.AbortDeformation(sReason:=EC_Print.ecPaStartErr.Desc, Src:=_pEcSrc^, bHideLog:=FALSE);
      Release(_pAttachedCt^);
		END_IF
  ELSIF _bPaStarted THEN
    //Release container when all points have been processed
    IF fbPa.bDone OR fbPa.bStop THEN
      _bPaStarted := FALSE;
      Release(_pAttachedCt^);
    (*ELSIF fbpa.bError THEN
      _pNewAttached^.AbortDeformation(sReason:=EC_Print.ecPaPrintErr.Desc, Src:=_pEcSrc^, bHideLog:=FALSE);
      Release(_pAttachedCt^);*)
    END_IF 
	END_IF
END_IF  

bPrintActive := _bPaStarted;

(*Logging config*)
fbPa.LogLevel := LogLevel;
fB_PcAdapter.LogLevel := LogLevel;
END_METHOD

END_FUNCTION_BLOCK

// ---- POUs/Print/DefGrid/FB_WorkerDefGrid_Python.TcPOU
{attribute 'reflection'} 
FUNCTION_BLOCK FB_WorkerDefGrid_Python EXTENDS FB_WorkerDefGrid IMPLEMENTS I_DeformationHandler
VAR_INPUT
END_VAR
VAR_OUTPUT
END_VAR
VAR
  // interface to py script
  fbPythonInterface : FB_PythonInterface;
  // references
  _iParamMediator : I_ParamMediator;
  
  // local copy of settings
  _bNewJob : BOOL;  // new job was activated
  _CamGridSettings : ST_CameraGridSettings;
  _DefGridSettings : ST_DefGridSettings;
  
  // local copy of job setting
  _aJobName         : T_MaxString;
  _aJobGuid         : T_MaxString;
  _fImageWidthM     : LREAL;          // image width in [m]
  _fImageDepthM     : LREAL;          // image depth in [m]
  

  // messages
  fbMsg_PythonNotRunning : FB_MESSAGE;
END_VAR

VAR CONSTANT
  fC_DEFAULT_WOKER_POSITION : LREAL := 0.01;      // default worker position in [m]
END_VAR

METHOD PROTECTED  Attach : BOOL
VAR_INPUT
  iCT              : I_CT;                         (*container at triggered event position*)
END_VAR
Attach := FALSE;
IF SUPER^.Attach(iCT:=iCT) THEN
  // OK, attached (enabled, was ok to be attached)
  IF _pNewAttached = 0 THEN RETURN; END_IF
  
  // setup check
  IF _iParamMediator = 0 THEN Release(iCT:=iCT); LogError('Invalid param mediator'); RETURN; END_IF
  
  // Additional worker checks
  // - do we have a valid job? used mode?
  IF _CamGridSettings.eCameraMode > E_CameraMode.NoCorrection AND (iCT.pJob = 0 OR NOT _bJobActive) THEN
    _pNewAttached^.AbortDeformation(sReason:='No valid job', Src:=_pEcSrc^, bHideLog:=FALSE);
     Release(iCT:=iCT);
     
  ELSIF _CamGridSettings.eCameraMode > E_CameraMode.NoCorrection THEN
    // OK attach
    // -- only create ct if a deformation is active
    IF CreateDefCt(iCT:=iCT) THEN
        // set state
        _pNewAttached^.StartScript(iDeformationHandler:=THIS^);
        // attached
        Attach := TRUE;
    END_IF
  ELSE
    ; // ignore attach
  END_IF
ELSE
  // parent attach failed
END_IF
END_METHOD

(*
  Create/Release virtual ct in deformation handlers.
  :return: TRUE if success
*)
METHOD PRIVATE CreateDefCt : BOOL;
VAR_INPUT
  iCT : I_CT;
END_VAR
IF iCT = 0 THEN RETURN; END_IF

IF _CamGridSettings.eCameraMode >= E_CameraMode.Live THEN
  IF fbPythonInterface.RegisterCT(iCT.pCT^.nMemIndex) THEN
    CreateDefCt := TRUE;
  ELSE
    _pAttachedCt^.AbortDeformation(sReason:='Could not register to script', Src:=_pEcSrc^, bHideLog:=FALSE);
  END_IF
ELSE
  CreateDefCt := TRUE;
END_IF
END_METHOD

METHOD DeleteCachedCt : BOOL
VAR_INPUT
	iCT	: I_CT;
END_VAR
DeleteDefCt(iCT:=iCT);
END_METHOD

(*
  Delete/Release virtual ct in deformation handlers.
  :return: TRUE if sucess
*)
METHOD DeleteDefCt : BOOL
VAR_INPUT
  iCT : I_CT;
END_VAR
IF iCT = 0 THEN RETURN; END_IF

IF _CamGridSettings.eCameraMode >= E_CameraMode.Live THEN
  IF fbPythonInterface.RemoveCT(iCT.pCT^.nMemIndex) THEN
    DeleteDefCt := TRUE;
  ELSE
    LogError('Could not delete ct in script');
  END_IF
END_IF
END_METHOD

METHOD Init
VAR_INPUT
  pMsgConfig : POINTER TO ST_MSG_CONFIG;         // message config
  fPrintResolution : LREAL := 1;                 // print(head) resolution in [dpi]
  fSubPxResolution : LREAL := 1;                 // SubPixel resolution [SubPx], resolution factor (fI_PrintResolution*fI_SubPxResolution=>Output resolution)
  bParallelCT : BOOL;                            // Support parallel processing of CTs
END_VAR
SUPER^.Init(pMsgConfig:=pMsgConfig, fPrintResolution:=fPrintResolution, fSubPxResolution:=fSubPxResolution, bParallelCT:=bParallelCT);

// Init messages
fbMsg_PythonNotRunning.pI_MsgConfig := _pMsgConfigExt;
fbMsg_PythonNotRunning.iI_MsgLocation := TO_INT(ePr_BLK_PU);
fbMsg_PythonNotRunning.iI_MsgNumber := eC_STAG_DEF_SCRIPT_NOT_RUNNING;
END_METHOD

METHOD InitWorkerPython
VAR_INPUT
  aScriptPath : T_MaxString;                     // path to cmd scripts
  //aAmsLocalHost : T_AmsNetID;                    // Ams netId localhost of the pc to run the script
  iDefGridParamMediator : I_ParamMediator;
END_VAR
IF NOT bInitialized OR _pCTM = 0 THEN LogError('Base Worker not initialized! call init() before'); RETURN; END_IF
IF iDefGridParamMediator = 0 THEN bInitialized := FALSE; LogError('Invalid parameter, no valid param mediator'); RETURN; END_IF

// worker specific init
_iParamMediator := iDefGridParamMediator;

fbPythonInterface.Init(
  sCTManagerPath := _pCTM^.sCTDefGridInstancesPath, 
  sScriptPath:=aScriptPath
);
END_METHOD

METHOD mJobStart
VAR_INPUT
	sJobDef	: CalmarCompPrint.I_JobDefinition;
END_VAR
// checks and fix defaults
IF _iParamMediator = 0 THEN LogError('JobStart: invalid parameter configuration'); RETURN; END_IF
IF _fWorkerPosition = 0 THEN _fWorkerPosition := fC_DEFAULT_WOKER_POSITION; LogError(F_Concat3(_name, ': worker position not set, set default=', TO_STRING(fC_DEFAULT_WOKER_POSITION))); END_IF

// configure
_aJobName := sJobDef.aJobName;
_aJobGuid := sJobDef.aJobId;
_fImageDepthM := sJobDef.fImageDepth/1000;
_fImageWidthM := sJobDef.fImageWidth/1000;

_bNewJob := TRUE;
_bJobActive := TRUE;
END_METHOD

METHOD  mJobStop
VAR_INPUT
	sStatus	: CalmarCompPrint.I_JobStatus;
END_VAR
fbPythonInterface.JobStop();
_bJobActive := FALSE;
END_METHOD

METHOD  work
VAR_INPUT
END_VAR
VAR
  i : UDINT;
  tempCt  : POINTER TO FB_ContainerDefGrid;
  bDeformationDone : BOOL;
  bDeformationError : BOOL;
END_VAR
VAR_INST
  rT_EnablePyIf  : R_TRIG;
END_VAR
SUPER^.work();

IF _iParamMediator = 0 THEN F_Report_Error(ErrType:=EN_REPORT_ERROR_TYPE.Report_Error_0Pointer); RETURN; END_IF
_CamGridSettings := _iParamMediator.sCameraGridSettings;
_DefGridSettings := _iParamMediator.sDeformationGridSettings;

// reconfig script after job started (Mediator parameter are defined in JobStart())
IF _bNewJob OR rT_EnablePyIf.Q THEN   // new job activated or re-enabled
  _bNewJob := FALSE;
  
  // setup script
  fbPythonInterface.JobStart(
    aJobName:=_aJobName,
    aJobGuid:=_aJobGuid,
    nJobImageWidth:=DINT_TO_UDINT(F_MeterToSubPixel(fPosMeter:=_fImageDepthM, fResoSubPx:=_fPrintResolution)),
    nJobImageHeigth:=DINT_TO_UDINT(F_MeterToSubPixel(fPosMeter:=_fImageWidthM, fResoSubPx:=_fPrintResolution)),
    nCamFrameWidth:=DINT_TO_UDINT(FC_LREAL_TO_DINT(_CamGridSettings.fGridFeaturePitch)),
    pGridSettings:=ADR(_DefGridSettings)
  );
END_IF

// start/stop script
IF _CamGridSettings.eCameraMode >= E_CameraMode.Live AND THIS^.bWorkerEnable THEN 
  fbPythonInterface.bEnable := TRUE;
ELSE
  fbPythonInterface.bEnable := FALSE;
END_IF
rT_EnablePyIf(CLK:=fbPythonInterface.bEnable);

fbPythonInterface();

IF _pAttachedCt <> 0 THEN
  // nothing to do anymore just release CT
  // NOTE: the delete of the CT is done by DeleteDefCt() method directly into fbPythonInterface
  Release(_pAttachedCt^);
END_IF

// messages
fbMsg_PythonNotRunning(bI_Status:=fbPythonInterface.bError);
IF fbMsg_PythonNotRunning.bMsgAck THEN fbPythonInterface.ackError(); END_IF
END_METHOD

END_FUNCTION_BLOCK

// ---- POUs/Print/DefGrid/FB_WorkerDefGrid_Verify.TcPOU
FUNCTION_BLOCK FB_WorkerDefGrid_Verify EXTENDS FB_WorkerDefGrid
VAR_OUTPUT
  bWateGateActive   AT%Q* : BOOL;     //  wate gate activation pulse
END_VAR
VAR
  bLastEject   : BOOL;   // stores state if last CT TRUE:=Eject, FALSE:=OK
  tpEjectPulse  : TP := (PT:=T#80MS);
  
  // print manager reference
  _pPm : POINTER TO FB_ProdManager_DMAX;
  
  // view verify history
  tpShowResult : TP := (PT:=T#700MS);
  nStateHistory : ARRAY[1..20] OF UINT;   // 2=???, 1=Eject, 0=OK
  nStateHistory_FillColor : ARRAY[1..20] OF UDINT;
  sResultText : STRING;
  
  // Grid Table export
  nCTId : DINT;
  bEnableGridExport : BOOL;
  nExportWrites : UDINT;
  sOutputPath : T_MaxString := 'C:\GridExport';
  sFileFormat : STRING := 'json';
  fbGridExporter : FB_GridDataExporter;
END_VAR

METHOD PROTECTED  Attach : BOOL
VAR_INPUT
  iCT              : I_CT;                         (*container at triggered event position*)
END_VAR
VAR 
  bSuccess         : BOOL;
END_VAR
IF SUPER^.Attach(iCT:=iCT) THEN
  
  // do CT supervision here and decice what happens with this sheet
   bSuccess := TRUE;
  IF NOT iCT.bValid AND iCT.bProductPresent AND iCT.pJob <> 0 THEN
    bSuccess := FALSE;
    // tag for ejection
    iCT.pCT^.lPrOutput := EN_PrinterOutput.trash;
	END_IF

  // finish CT in production
  IF _pPm <> 0 THEN 
    _pPm^.CT_Finish(sCT:=iCT, bSuccess:=bSuccess);      // report to job status
  ELSE
    LogError('PrintManager not set');
	END_IF
  
  // select output
  IF iCT.pCT^.lPrOutput = EN_PrinterOutput.trash THEN
    // create eject trigger
    tpEjectPulse(IN:=TRUE);
    bLastEject := TRUE;
    LogLvl(Lvl:=E_LogSeverity.Debug, Msg:=F_Concat2('Eject CT: ', _pAttachedCt^.print(0)));
  ELSE
    tpEjectPulse(IN:=FALSE);
    bLastEject := FALSE;
	END_IF
  
  // History view
  MEMMOVE(destAddr:=ADR(nStateHistory[1+1]),           srcAddr:=ADR(nStateHistory[1]),           n:=((SIZEOF(nStateHistory)/SIZEOF(nStateHistory[1]))-1)*SIZEOF(nStateHistory[1]));
  MEMMOVE(destAddr:=ADR(nStateHistory_FillColor[1+1]), srcAddr:=ADR(nStateHistory_FillColor[1]), n:=((SIZEOF(nStateHistory_FillColor)/SIZEOF(nStateHistory_FillColor[1]))-1)*SIZEOF(nStateHistory_FillColor[1]));
  
  nStateHistory[1] := SEL(bLastEject=TRUE, 0, 1);
  sResultText := SEL(bLastEject=TRUE, 'OK', 'NOK');

  IF iCT.bProductPresent AND iCT.bValid THEN        nStateHistory_FillColor[1] := 16#FF000000 OR WebColors.LightGreen.lCode;
  ELSIF iCT.bProductPresent AND NOT iCT.bValid AND iCT.pCT^.lPrOutput = EN_PrinterOutput.trash THEN nStateHistory_FillColor[1] := 16#FF000000 OR WebColors.LightSalmon.lCode;   
  ELSIF iCT.bProductPresent AND NOT iCT.bValid AND iCT.pCT^.lPrOutput <> EN_PrinterOutput.trash THEN nStateHistory_FillColor[1] := 16#FF000000 OR WebColors.LightGray.lCode;
	ELSIF NOT iCT.bProductPresent THEN                nStateHistory_FillColor[1] := 16#FF000000 OR WebColors.LightGray.lCode;
  END_IF

  tpShowResult(IN:=FALSE);
  tpShowResult(IN:=TRUE);
  
  // grid history
  IF bEnableGridExport AND iCT.bProductPresent AND nExportWrites < 100 THEN
    nCTId := _pAttachedCt^.pCT^.iId;
    sFileFormat := SEL(sFileFormat='csv', 'json', 'csv');
    fbGridExporter(
        sOutputDir:=sOutputPath,
        sFileName:=F_Concat4('\Export_', TO_STRING(nCTId), '.', sFileFormat),
        pFbImageDeformation:=_pAttachedCt^.pImageDeformation,
        //nSelectGrid:=
    );
    fbGridExporter.startExport();
    nExportWrites:=nExportWrites+1;
  ELSE
    nExportWrites := 0; bEnableGridExport := FALSE;
  END_IF
END_IF
END_METHOD

(*
  Set PrintManager.
*)
METHOD InitWorkerVerify : BOOL
VAR_INPUT
  pPm : POINTER TO FB_ProdManager_DMAX;
END_VAR
IF pPm = 0 THEN LogError('Invalid Pm given'); END_IF

_pPm := pPm;  // register print manager reference
END_METHOD

METHOD   mJobStart
VAR_INPUT
	sJobDef	: CalmarCompPrint.I_JobDefinition;
END_VAR
END_METHOD

METHOD  mJobStop
VAR_INPUT
	sStatus	: CalmarCompPrint.I_JobStatus;
END_VAR
END_METHOD

METHOD Release : BOOL
VAR_INPUT
  iCT              : I_CT;                         (*container at triggered event position*)
END_VAR
IF SUPER^.Release(iCT := iCT) THEN
  ;
END_IF
END_METHOD

METHOD  work
VAR_INST
  fT_Pulse  : F_TRIG;
END_VAR
SUPER^.work();

// output signal handling
tpEjectPulse(Q=>bWateGateActive);
fT_Pulse(CLK:=bWateGateActive);
tpShowResult();
//IF tpShowResult.IN:=TRUE AND NOT tpShowResult.Q THEN tpShowResult(IN:=FALSE); END_IF   // reset pulse

fbGridExporter();

// release
IF tpEjectPulse.IN THEN
  IF fT_Pulse.Q THEN  
    tpEjectPulse(IN:=FALSE);
  END_IF
END_IF

IF _pAttachedCt <> 0 THEN   // just release any attached container in this cycle
  Release(iCT:=_pAttachedCt^);
END_IF
END_METHOD

END_FUNCTION_BLOCK

// ---- POUs/Print/FB_SheetDetectSupervision.TcPOU
FUNCTION_BLOCK FB_SheetDetectSupervision
VAR_INPUT
  IbSensorSheetCalender                   AT%I* : BOOL;            // Sensor signal B250
  IbSensorSheetInlet                      AT%I* : BOOL;            // Sensor signal B257
  IbSensorSheetOutlet                     AT%I* : BOOL;            // Sensor signal B254

  InCurrentPos                                  : DINT;            // Current position in [SubPx]
  IbMachineStopped                              : BOOL;            // Machine stopped
  IbInhibitSheetTrigger                         : BOOL;            // inhibit trigger signals for substrate length
  IbCameraTrigger                               : BOOL;            // Camera trigger
END_VAR

VAR_OUTPUT
  ObSheetJamPrintingSystem                AT%Q* : BOOL;            // Sheet jam in printing system detected

  ObCameraTriggerEnable                         : BOOL;            // Camera trigger enable
  ObCameraTriggerIncorrect                      : BOOL;            // Camera trigger incorrect
  ObCameraTriggerSupervison                     : BOOL;            // Camera trigger supervision for sheet jam
  ObSheetDetectFree                             : BOOL;            // sheet detect sensors are free
END_VAR

VAR
  _PrintSubPixelResolution                      : UDINT := 600 * 32;           // Print sub pixel resolution

  fbSheetDetectRingbuffer01                     : FB_RINGBUFFER;
  fbSheetDetectRingbuffer02                     : FB_RINGBUFFER;

  rfTrig_CameraTriggerSupervison                : RF_TRIG;
  bCameraTriggerSupervisonOn                    : BOOL;
  
  rfTrig_MachineStopped                         : RF_TRIG;

  // jam event
  rTrig_SheetJam                                : R_TRIG;
  _bSheetJamEvent                               : BOOL;
  
  // error handling 
  nConversionErrorCounter                       : UDINT;
END_VAR

VAR PERSISTENT
  RemSheetDetectSupervisionPar                  : ST_SheetDetectSupervisionPar;
END_VAR

rfTrig_MachineStopped(CLK := IbMachineStopped);

(*B250 => B256*)
fbSheetDetectRingbuffer01.pI_ConversionErr      := ADR(nConversionErrorCounter);
fbSheetDetectRingbuffer01.bI_Reset              := IbMachineStopped;
fbSheetDetectRingbuffer01.bI_Sensor             := NOT IbSensorSheetCalender;
fbSheetDetectRingbuffer01.iI_CurrentPos         := DINT_TO_UDINT(InCurrentPos);
fbSheetDetectRingbuffer01.iI_Pg_Offset          := 0;
fbSheetDetectRingbuffer01.iI_Offset_X0          := fbSheetDetectRingbuffer01.iI_CurrentPos + DINT_TO_UDINT(F_MeterToSubPixel(RemSheetDetectSupervisionPar.fR_SheetDetectDistance01, UDINT_TO_LREAL(_PrintSubPixelResolution)));           
fbSheetDetectRingbuffer01.iI_Resolution         := UDINT_TO_INT(_PrintSubPixelResolution);
fbSheetDetectRingbuffer01.fI_ShiftDistance      := 0 - RemSheetDetectSupervisionPar.fR_SheetDetectRange01_m;
fbSheetDetectRingbuffer01();

(*B256 => B254*)
fbSheetDetectRingbuffer02.pI_ConversionErr      := ADR(nConversionErrorCounter);
fbSheetDetectRingbuffer02.bI_Reset              := IbMachineStopped;
fbSheetDetectRingbuffer02.bI_Sensor             := IbCameraTrigger;
fbSheetDetectRingbuffer02.iI_CurrentPos         := DINT_TO_UDINT(InCurrentPos);
fbSheetDetectRingbuffer02.iI_Pg_Offset          := 0;
fbSheetDetectRingbuffer02.iI_Offset_X0          := fbSheetDetectRingbuffer02.iI_CurrentPos + DINT_TO_UDINT(F_MeterToSubPixel(RemSheetDetectSupervisionPar.fR_SheetDetectDistance02, UDINT_TO_LREAL(_PrintSubPixelResolution)));           
fbSheetDetectRingbuffer02.iI_Resolution         := UDINT_TO_INT(_PrintSubPixelResolution);
fbSheetDetectRingbuffer02.fI_ShiftDistance      := 0 - RemSheetDetectSupervisionPar.fR_SheetDetectRange02_m;
fbSheetDetectRingbuffer02();

RemSheetDetectSupervisionPar.nR_SheetDetectRange01_SubPx := F_MeterToSubPixel(REAL_TO_LREAL(RemSheetDetectSupervisionPar.fR_SheetDetectRange01_m), UDINT_TO_LREAL(_PrintSubPixelResolution));
RemSheetDetectSupervisionPar.nR_SheetDetectRange02_SubPx := F_MeterToSubPixel(REAL_TO_LREAL(RemSheetDetectSupervisionPar.fR_SheetDetectRange02_m), UDINT_TO_LREAL(_PrintSubPixelResolution));

IF RemSheetDetectSupervisionPar.bR_Enable THEN
  (*Masking sheet detection of camera system*)
  ObCameraTriggerEnable     :=     (InCurrentPos > (fbSheetDetectRingbuffer01.iO_ShiftOffset_X0 - RemSheetDetectSupervisionPar.nR_SheetDetectRange01_SubPx)) 
                               AND (InCurrentPos < (fbSheetDetectRingbuffer01.iO_ShiftOffset_X0 + RemSheetDetectSupervisionPar.nR_SheetDetectRange01_SubPx));
  (*Sheet trigger was incorrect because of faulty detection*)
  IF NOT ObCameraTriggerEnable AND IbSensorSheetInlet AND NOT IbInhibitSheetTrigger THEN
    ObCameraTriggerIncorrect := TRUE;
  END_IF

  (*Sheet jam supervision*)
  ObCameraTriggerSupervison :=     (InCurrentPos > (fbSheetDetectRingbuffer02.iO_ShiftOffset_X0 - RemSheetDetectSupervisionPar.nR_SheetDetectRange02_SubPx)) 
                               AND (InCurrentPos < (fbSheetDetectRingbuffer02.iO_ShiftOffset_X0 + RemSheetDetectSupervisionPar.nR_SheetDetectRange02_SubPx));
  rfTrig_CameraTriggerSupervison(CLK := ObCameraTriggerSupervison);
  IF rfTrig_CameraTriggerSupervison.RT THEN
    bCameraTriggerSupervisonOn := TRUE;
  END_IF
  IF bCameraTriggerSupervisonOn AND IbSensorSheetOutlet THEN
    bCameraTriggerSupervisonOn := FALSE;
  END_IF
  IF rfTrig_CameraTriggerSupervison.FT AND bCameraTriggerSupervisonOn THEN
    ObSheetJamPrintingSystem   := TRUE;
    bCameraTriggerSupervisonOn := FALSE;
  END_IF

  ObSheetDetectFree := TRUE;
  IF IbMachineStopped THEN
    ObCameraTriggerIncorrect   := FALSE;
    bCameraTriggerSupervisonOn := FALSE;

    IF NOT IbSensorSheetCalender OR IbSensorSheetInlet OR IbSensorSheetOutlet THEN
      ObSheetDetectFree := FALSE;
    END_IF
  END_IF
  IF rfTrig_MachineStopped.FT THEN
    ObSheetJamPrintingSystem   := FALSE;
  END_IF
ELSE
  ObCameraTriggerEnable     := TRUE;
  ObCameraTriggerIncorrect  := FALSE;
  ObSheetJamPrintingSystem  := FALSE;
  ObSheetDetectFree         := TRUE;
END_IF

rTrig_SheetJam(CLK:=ObSheetJamPrintingSystem);
IF rTrig_SheetJam.Q THEN _bSheetJamEvent := TRUE; END_IF

PROPERTY bSheetJamEvent : BOOL
GET
bSheetJamEvent := _bSheetJamEvent;
_bSheetJamEvent := FALSE;
END_GET
END_PROPERTY

PROPERTY PrintSubPixelResolution : UDINT
SET
_PrintSubPixelResolution := PrintSubPixelResolution;
END_SET
END_PROPERTY

END_FUNCTION_BLOCK

// ---- GlobalTextList.TcGTLO
TEXTLIST GlobalTextList
  10210 = '  x:%0.5f'
  6570 = '  y:%0.5f'
  781 = ' Camera offset Y [mm]: %f'
  2961 = ' cM: Camera start margin [m]: %f'
  5665 = ' Modus: %s'
  13668 = ' Nb teach marks: %d'
  13672 = ' Nb teach sectors: %d'
  9596 = ' Number of marks: %d'
  10437 = ' pW: Actual PrintUnit width [m]: %f'
  8296 = ' pWc: PrintUnit width [m]: %f'
  2948 = ' Sector of transmission: %d'
  5660 = ' Version number: %d'
  1184 = '%0.01f'
  14098 = '%0.02f'
  4085 = '%0.02f m/s'
  13676 = '%0.04f'
  8040 = '%0.06f'
  303 = '%0.0f'
  2502 = '%0.0f [m]'
  8178 = '%0.0f [px]'
  293 = '%0.1f'
  11885 = '%0.1f [cols]'
  430 = '%0.1f [m/min]'
  941 = '%0.1f [um]'
  10 = '%0.2f'
  993 = '%0.3f'
  1945 = '%0.3f [m/min]'
  6769 = '%0.3f [m/s]'
  4949 = '%0.3f [ms]'
  10891 = '%0.3f [m]'
  7216 = '%0.3f [px]'
  1864 = '%0.4f'
  11719 = '%0.4f  [m]'
  1796 = '%0.4f [ms]'
  7315 = '%0.4f [m]'
  1072 = '%0.5f'
  1822 = '%0.5f [m]'
  1887 = '%0.6f [m/s]'
  1147 = '%0.6f [ms]'
  820 = '%0.6f [m]'
  2289 = '%0.6f [um]'
  704 = '%1.1f'
  3079 = '%1.1f mm'
  3009 = '%1.1f mm/s'
  1930 = '%1.2f'
  741 = '%1.2f mm'
  3014 = '%1.3f mm'
  2489 = '%1.3f [mm]'
  6533 = '%1.3f [px]'
  3085 = '%1.4f m'
  7362 = '%1.4f [ms]'
  2560 = '%1.4f [m]'
  3481 = '%1.5f [m]'
  9 = '%d'
  3602 = '%d [px]'
  2955 = '%d [um]'
  456 = '%f'
  2383 = '%f [m/min]'
  5388 = '%f [mm]'
  812 = '%f [m]'
  2912 = '%f [s.p.min]'
  3959 = '%f [um]'
  27 = '%s'
  260 = '%s%%'
  9843 = '(Hw)Enable'
  3930 = '(not used) CameraToPrintUnit'
  17381 = '(viratual) generated'
  12232 = '*'
  447 = '+'
  7024 = '+/- %0.4f'
  8411 = '-'
  68 = '/'
  2589 = '1'
  2552 = '1. Activate (Drop)SpeedComp with Time set to 0\n\n2. Test print with production speed1\n   -> Measure displacement with Speed1\n\n3. Test print with production speed2\n   -> Measure displacement with Speed2\n\n4. Enter Speed and Displacement values in\n    table for Test1 and Test2\n\n5. Start new Time calculation'
  245 = '1. Activate (Drop)SpeedComp with Time set to 0\n\n2. Test print with Speed1\n   -> Measure displacement with Speed1\n\n3. Test print with Speed2\n   -> Measure displacement with Speed2\n\n4. Enter Speed and Displacement values in\n    table for Test1 and Test2\n\n5. Start new Time calculation'
  864 = '1. Activate (Drop)SpeedComp with Time set to 0\n\n2. Test1 print with production speed1\n   -> Measure displacement with Speed1\n\n3. Test2 print with production speed2\n   -> Measure displacement with Speed2\n\n4. Enter Speed and Displacement values in\n    table for Test1 and Test2\n\n5. Start new Time calculation'
  835 = '1. Activate (Drop)SpeedComp with Time set to 0\n\n2. Test1: print with production speed1\n   -> Measure displacement with Speed1\n\n3. Test2: print with production speed2\n   -> Measure displacement with Speed2\n\n4. Enter Speed and Displacement values in\n    table for Test1 and Test2\n\n5. Start new Time calculation'
  41 = '1. Activate DropSpeeCmp'
  1428 = '1. Activate DropSpeeComp\n   + Set Time to 0'
  1322 = '1. Activate DropSpeeComp\n   + Set Time to 0\n\n\n\n'
  1646 = '1. Activate DropSpeeComp\n   + Set Time to 0\n\n2. Test print with Speed1\n   + Measure displacement with Speed1\n\n'
  478 = '1. Activate DropSpeeComp\n   + Set Time to 0\n\n2. Test print with Speed1\n   + Measure displacement with Speed1\n\n3. Test print with Speed2\n   + Measure displacement with Speed2\n'
  2206 = '1. Activate DropSpeeComp\n   + Set Time to 0\n\n2. Test print with Speed1\n   + Measure displacement with Speed1\n\n3. Test print with Speed2\n   + Measure displacement with Speed2\n\n\n4. Enter values in table for Test1 and Test2\n\n5. Start new Time calculation'
  543 = '1. Activate DropSpeeComp\n   + Set Time to 0\n\n2. Test print with Speed1\n   + Measure displacement with Speed1\n\n3. Test print with Speed2\n   + Measure displacement with Speed2\n\n\n\n4. Enter values in table for Test1 and Test2'
  1417 = '1. Activate DropSpeeComp\n   + Set Time to 0\n\n2. Test print with Speed1\n   + Measure displacement with Speed1\n\n3. Test print with Speed2\n   + Measure displacement with Speed2\n\n5. Start new Time calculation\n\n4. Enter values in table for Test1 and Test2'
  2118 = '1. Activate DropSpeeComp\n   Set Time to 0'
  1160 = '1. Activate DropSpeeComp with Time set to 0\n\n2. Test print with Speed1\n   + Measure displacement with Speed1\n\n3. Test print with Speed2\n   + Measure displacement with Speed2\n\n\n4. Enter values in table for Test1 and Test2\n\n5. Start new Time calculation'
  1763 = '1. Activate DropSpeeComp with Time set to 0\n\n2. Test print with Speed1\n   + Measure displacement with Speed1\n\n3. Test print with Speed2\n   + Measure displacement with Speed2\n\n4. Enter values in table for Test1 and Test2\n\n5. Start new Time calculation'
  1928 = '1. Activate DropSpeeComp with Time set to 0\n\n2. Test print with Speed1\n   -> Measure displacement with Speed1\n\n3. Test print with Speed2\n   -> Measure displacement with Speed2\n\n4. Enter Speed and Displacement values\n     in table for Test1 and Test2\n\n5. Start new Time calculation'
  2230 = '1. Activate DropSpeeComp with Time set to 0\n\n2. Test print with Speed1\n   -> Measure displacement with Speed1\n\n3. Test print with Speed2\n   -> Measure displacement with Speed2\n\n4. Enter Speed and Displacement values in\n    table for Test1 and Test2\n\n5. Start new Time calculation'
  2617 = '1. Activate DropSpeeComp with Time set to 0\n\n2. Test print with Speed1\n   -> Measure displacement with Speed1\n\n3. Test print with Speed2\n   -> Measure displacement with Speed2\n\n4. Enter Speed and Displacement values in     table for Test1 and Test2\n\n5. Start new Time calculation'
  167 = '1. Activate DropSpeeComp with Time set to 0\n\n2. Test print with Speed1\n   -> Measure displacement with Speed1\n\n3. Test print with Speed2\n   -> Measure displacement with Speed2\n\n4. Enter Speed and Displacement values in table for Test1 and Test2\n\n5. Start new Time calculation'
  1944 = '1. Activate DropSpeeComp with Time set to 0\n\n2. Test print with Speed1\n   -> Measure displacement with Speed1\n\n3. Test print with Speed2\n   -> Measure displacement with Speed2\n\n4. Enter values in table for Test1 and Test2\n\n5. Start new Time calculation'
  363 = '1. Activate DropSpeedComp with Time set to 0\n\n2. Test print with Speed1\n   -> Measure displacement with Speed1\n\n3. Test print with Speed2\n   -> Measure displacement with Speed2\n\n4. Enter Speed and Displacement values in\n    table for Test1 and Test2\n\n5. Start new Time calculation'
  2048 = '1. Active DropSpeedComp'
  2104 = '1. Set Time to 0'
  7016 = '2*a'
  1505 = '2. Test print with Speed1\n   + Measure displacement with Speed1'
  2308 = '2. Test print with Speed1\n   Measure displacement with Speed1'
  1658 = '3. Test print with Speed2\n   + Measure displacement with Speed2'
  77 = '3. Test print with Speed2\n   Measure displacement with Speed2'
  550 = '4. Calculate new Time'
  581 = '4. Enter values in table for Test1 and Test2'
  1286 = '4. Start new Time calculation'
  2168 = '4p PLC'
  739 = '5. Start new Time calculation'
  8190 = '<'
  11083 = '<-'
  448 = '='
  6003 = '>'
  9654 = '>Camera(s)'
  1163 = '>FineAlignement'
  15769 = '>PrintPosition'
  18969 = '>WorkerPrint PG1 (Row1)'
  2212 = '>WorkerPrint PG2 (Row2)'
  19156 = 'a'
  14960 = 'a (mark size)'
  3758 = 'a/2'
  7335 = 'a: %d'
  4185 = 'Abort'
  3571 = 'Acknowledge'
  1383 = 'Act pos.'
  140 = 'Active'
  1300 = 'active camera device'
  517 = 'active camera device type'
  7324 = 'active camera mode'
  2160 = 'Actual Y-Resolution [dpi]: %1.4f'
  8699 = 'added points'
  1427 = 'ADS axis position'
  590 = 'ADS Axis Position'
  5009 = 'ADS command'
  717 = 'ADS Commands'
  9674 = 'ADS PG shift'
  2259 = 'ADS PU shift'
  4169 = 'ADS settings'
  723 = 'ADS Settings'
  15944 = 'All Epsitron'
  3353 = 'All Epsitron OK'
  5267 = 'All Inputs ok'
  5680 = 'AnalogMaxDigit'
  3775 = 'Auto'
  671 = 'AUTO/MANU CONTROL'
  4177 = 'Automatic Mode'
  1339 = 'Automatic or ManualTeach'
  2606 = 'AutomaticMode or ManualTeach'
  12039 = 'b'
  7246 = 'b (mark size)'
  9731 = 'B250'
  2262 = 'B254'
  16217 = 'B257'
  2111 = 'Back'
  608 = 'Bacl'
  3856 = 'bStopReady'
  210 = 'Busy'
  19400 = 'by calculation'
  6619 = 'C'
  411 = 'c'
  9048 = 'c (mark distance)'
  744 = 'C1'
  743 = 'C2'
  1065 = 'c: %d'
  3129 = 'c:%d'
  710 = 'Ca/Pu'
  136 = 'Calculate new time'
  1431 = 'Calculate new Time'
  13216 = 'Calender'
  6811 = 'cam simulation'
  1299 = 'Cam valid'
  1186 = 'Cam Valid'
  4259 = 'Camera'
  13991 = 'Camera activated'
  11573 = 'Camera Detail: %s'
  1141 = 'Camera ip address'
  1321 = 'camera mode desired'
  530 = 'camera mode desired (active cam)'
  1086 = 'Camera name'
  1061 = 'camera port'
  2103 = 'Camera sink'
  6170 = 'Camera temperature [°C]: %1.1f'
  5051 = 'Camera trigger'
  1990 = 'Camera type'
  9680 = 'Camera->PU'
  11139 = 'CameraToPrintUnit'
  8862 = 'CameraTrigger'
  14480 = 'CamPointsFifo'
  5607 = 'CamToPU'
  5019 = 'CanEx'
  7354 = 'cfb'
  10808 = 'Charged columns'
  8294 = 'Check delay'
  708 = 'Clean'
  3790 = 'Clean Active'
  719 = 'Clean after Capping'
  720 = 'Clean after Purge'
  1935 = 'Clean Head'
  1246 = 'Clean head (max %d)'
  711 = 'Clean Unit'
  15882 = 'Clean unit (max %d)'
  14428 = 'CleanCappPosition'
  4247 = 'CLEANER'
  4468 = 'Cleaner pump'
  265 = 'Cleaning'
  3760 = 'Cleaning Operations'
  740 = 'Cleaning Safe '
  4828 = 'CleaningProcess'
  212 = 'col'
  1396 = 'Column Precharge'
  6407 = 'Comp.'
  10565 = 'Compensation temperatur extension'
  11736 = 'configured camera mode, active=%s'
  10779 = 'Connected'
  9558 = 'constant'
  7336 = 'correction relative'
  6221 = 'csv'
  8478 = 'ct'
  3579 = 'CT'
  8221 = 'CT @Deformation (more corrections followed @Print!)'
  1165 = 'CT Id=%d'
  5554 = 'CT ImageDeformation'
  1850 = 'CT PrintRef'
  6824 = 'CT Status'
  17584 = 'CTDetail  @PrintWorker[1]  !No FineAlignment yet applied!'
  11030 = 'CTManager'
  15305 = 'Current'
  69 = 'current camera mode (active cam)'
  1219 = 'Current columen relative to Worker Attach'
  6060 = 'Current column'
  10240 = 'Current CT'
  10438 = 'Current position'
  10758 = 'Current reso used (from machine)'
  20158 = 'Current Speed'
  4981 = 'Current step'
  1573 = 'CurrentSpeed [m/s]'
  389 = 'D'
  2060 = 'Dead Time'
  1132 = 'Dead/Add Time'
  4013 = 'Dead/Add Time [ms]'
  21105 = 'Debug & Simulation'
  12899 = 'Deformation'
  1100 = 'DeformType'
  3003 = 'Delta P'
  2040 = 'Detect -> Cam'
  7545 = 'Detect -> Cam (Trig.Dist.)'
  18521 = 'Detected'
  6 = 'detected length [mm]'
  10000 = 'detected length [m]'
  1172 = 'Detected Marks: %d'
  9097 = 'Detection'
  10216 = 'Detection range [m]'
  12392 = 'DetectToCam'
  11747 = 'DetectToCamera'
  1597 = 'Device type'
  4990 = 'DevOpActive'
  5555 = 'Diff [mm]'
  8247 = 'Diff [m]'
  16644 = 'Direction'
  1171 = 'Disable left SLM'
  6432 = 'Disable right SLM'
  2162 = 'Displacement'
  1297 = 'Displacment'
  4696 = 'Distance in [p]'
  16193 = 'Distance [m]'
  4984 = 'DistBetweenMasks'
  3424 = 'DistToCamera'
  3798 = 'DO'
  152 = 'Done'
  1364 = 'Done LastMrk'
  4615 = 'DropSpeed'
  11858 = 'DropSpeed compensation'
  13254 = 'DropSpeed Compensation'
  1196 = 'DropSpeed Setup'
  4971 = 'DropSpeed [m/s]'
  3476 = 'DX'
  1038 = 'dx'
  8677 = 'dX (Global Deformation Shift)'
  1075 = 'dx (middle)'
  4842 = 'dX shift (points)'
  4026 = 'dx [mm]'
  6941 = 'dx [m]'
  15980 = 'dx:%0.5f'
  5761 = 'dx=%0.5f'
  1050 = 'DY'
  1039 = 'dy'
  10840 = 'dY (Global Deformation Shift)'
  2175 = 'dy [mm]'
  14658 = 'dy [m]'
  2520 = 'dy:%0.5f'
  15313 = 'dy=%0.5f'
  18481 = 'e state'
  2650 = 'Effective Encoder Resolution Detection'
  3372 = 'Effective[mm]'
  8187 = 'Effective[m]'
  5571 = 'Eject'
  4244 = 'Ejected'
  6817 = 'Ejected=1'
  2388 = 'EjectTriggerLength'
  3062 = 'EL7041'
  685 = 'EL7201'
  10657 = 'ElapsedTime: %s'
  4263 = 'Emergency stop'
  8 = 'Enable'
  2501 = 'Enable Correction'
  147 = 'Enable Speed Compensation'
  234 = 'Enabled'
  7765 = 'Enabled compensation'
  1980 = 'Encoder'
  7568 = 'Encoder Filter'
  4996 = 'encoder filter active'
  14488 = 'Encoder speed compensation factor'
  5880 = 'Encoder speed compensation reference speed'
  2208 = 'EncoderReso'
  9966 = 'EncoderResolution'
  6771 = 'EncSpeedCompFactor'
  9759 = 'EncSpeedCompRefSpeed'
  1636 = 'EncSpeedCorrection'
  417 = 'Endless'
  5930 = 'Engaged'
  714 = 'Enter Capping'
  688 = 'Epsitron Control'
  4621 = 'Err: %d'
  40 = 'Error'
  13934 = 'Error 0x%X'
  1158 = 'Error level'
  4543 = 'error: %d'
  731 = 'EStop'
  3722 = 'EStop Ok'
  4412 = 'exec'
  5028 = 'Exec'
  2082 = 'Execute device reset only in CU park position!'
  14686 = 'Execute device reset only in PU service position!'
  2569 = 'Execute device reset only in safe state'
  18335 = 'Exeeds max. speed=%f'
  11482 = 'Exhaust active'
  1734 = 'Exhaust system'
  2867 = 'Exhaust vacuum measurement 0-50mBar'
  715 = 'Exit Capping'
  3291 = 'Exporter'
  10708 = 'e_DeltaT'
  4278 = 'f (%d)'
  2541 = 'F=%d'
  1765 = 'Fast Stop Request'
  7021 = 'FastStop'
  1938 = 'Fault Acknowledge'
  11231 = 'Feature grid'
  17650 = 'FeatureGrid'
  4662 = 'feedback [mBar]'
  5376 = 'File Format'
  2633 = 'File Name'
  971 = 'File Path'
  3286 = 'filter active'
  682 = 'filter active (green)'
  12495 = 'Filter depth'
  1635 = 'filter=%d'
  2291 = 'Filters settings'
  705 = 'Force Close'
  9669 = 'Force DefGrid stream OFF'
  4095 = 'Force Grid OFF (gridPs=0)'
  729 = 'Force Open'
  12720 = 'ForceGrid OFF'
  3916 = 'Format'
  18523 = 'Format Machine'
  12999 = 'fPrintStartOffset'
  1948 = 'Frames for this image'
  1067 = 'From row: %d'
  913 = 'fsf'
  1148 = 'fsf\nsdfsd\nsdfsd'
  5979 = 'F[%d]'
  453 = 'Gap [mm]'
  1280 = 'Gap [m]'
  982 = 'Gap [m], %d [mm]'
  4929 = 'Global dX'
  1069 = 'Global dY'
  18887 = 'GlobalShift Dx/Dy'
  5637 = 'Grid Exporter'
  1397 = 'Grid ImageOffset Y [px]'
  12596 = 'Grid Points'
  7895 = 'Grid size c/r/y'
  851 = 'Grid Size X'
  1029 = 'Grid SizeY'
  6188 = 'GridPitch x/y'
  13281 = 'GridPoint history ->'
  15797 = 'GridPointsFifo'
  3068 = 'GridSel'
  5110 = 'h:%0.3f'
  15957 = 'h=%0.4f'
  5131 = 'Hardware'
  11305 = 'Head Gap [m]'
  5194 = 'Head Offset Plate [m]'
  1014 = 'History'
  12822 = 'Host: %s'
  2960 = 'HwEnable'
  388 = 'I'
  5854 = 'ID'
  1719 = 'id'
  18013 = 'Id'
  3111 = 'id of ct head'
  11673 = 'Idx'
  428 = 'Ign'
  597 = 'ignored'
  14585 = 'Image Height'
  9559 = 'Image Length'
  3696 = 'Image Length Job'
  425 = 'Image Width'
  2947 = 'ImageLength'
  4494 = 'ImageLength effect.'
  17474 = 'IMLen: %0.04f'
  12205 = 'IMWidth: %0.04f'
  733 = 'In     Out'
  6859 = 'InArea'
  9554 = 'Infeed'
  1262 = 'Inhibit trigger'
  15988 = 'Init'
  166 = 'Init ok'
  8950 = 'Initialized'
  9607 = 'InkQuantity'
  5070 = 'InPrintPos'
  3260 = 'Input (Fuse)'
  1115 = 'Inputs'
  3753 = 'Interlock'
  2159 = 'invalid & ignored marks'
  2281 = 'Invalid marks (ignored)'
  4159 = 'inverted'
  5409 = 'Inverted'
  6150 = 'inverted X'
  386 = 'Job'
  10238 = 'Job is active'
  1053 = 'JobActive'
  7197 = 'json'
  3174 = 'l'
  12184 = 'Len'
  2034 = 'Len Detect [mm]'
  2995 = 'Len Detected'
  8363 = 'LenghtMissmatch'
  3520 = 'Length check'
  18494 = 'Length Configured'
  14466 = 'Length diff'
  13542 = 'Length Effective'
  15936 = 'Length not in range'
  376 = 'Length [mm]'
  1522 = 'Length [m]'
  1876 = 'LenSq [mm]'
  267 = 'LenSq [m]'
  6355 = 'LenSquare'
  2735 = 'LenTr [mm]'
  14842 = 'LenTriangle'
  737 = 'LimitDN'
  4478 = 'Limits from machine'
  736 = 'LimitUP'
  15280 = 'LineCamera'
  18927 = 'Logger'
  11756 = 'LogLevel'
  8854 = 'Low intense mode'
  8103 = 'lsq=%0.4f'
  17552 = 'ltr=%0.4f'
  2934 = 'lx'
  2937 = 'ly'
  287 = 'm'
  3178 = 'm=%d'
  6479 = 'Machine Interface'
  1179 = 'MachineStopped'
  15 = 'Maintenance'
  3805 = 'MANU CONTROL'
  20108 = 'Manu Trigger'
  2076 = 'ManualTeach'
  539 = 'Mark at S1 invalid length'
  3844 = 'Mark at S1 too short'
  7032 = 'Mark at S2 invalid length'
  3478 = 'Mark at S2 too short'
  6031 = 'Mark Details'
  1296 = 'Mark History'
  1816 = 'Mark is flipped/inverted'
  15343 = 'Mark Lenght Margin'
  1191 = 'Mark length in [mm], minimum length=%0.02f [mm]'
  6077 = 'mark not proper detected'
  12613 = 'Mark per Use'
  9961 = 'Mark Settings'
  1952 = 'Mark teach'
  18681 = 'mark too short'
  16062 = 'MarkCamera'
  8898 = 'MarkDefinition'
  2476 = 'MarkDefinition Detail - Mark[%d]'
  20000 = 'MarkDetection'
  8025 = 'MarkDistFromCenter: %0.04f'
  9087 = 'marks valid'
  7504 = 'Master module idx'
  813 = 'MAV filter size "Dist in Pulse"'
  3301 = 'MAV filter size "Dist in Pulse" measured'
  12087 = 'MAV size "Dist in Pulse" measured'
  5710 = 'MAV size "Pulse Speed"'
  1189 = 'Max Limit'
  13601 = 'Max. Speed [m/s]'
  6002 = 'MaxMas'
  4885 = 'MaxMaster'
  516 = 'MaxModule'
  6815 = 'MaxPM'
  4790 = 'MaxSubstrate Factor'
  17117 = 'Measure: %d'
  12383 = 'MeasuredEncoderPulse'
  8147 = 'Measurement'
  19576 = 'Measurement aborted'
  12224 = 'measurement counter'
  22057 = 'Min Limit'
  16128 = 'Min. Speed'
  1173 = 'Min. Speed for Production'
  7865 = 'Min. speed production [m/min]'
  2019 = 'Min. Speed [m/s]'
  10619 = 'Min. Use Length'
  2528 = 'MinM'
  5381 = 'MinMa'
  6191 = 'MinMas'
  3216 = 'MinMaster'
  3134 = 'MinMstrer'
  2492 = 'MinProd'
  2310 = 'MinProd.'
  21567 = 'Mis'
  1193 = 'Missed'
  1120 = 'missed'
  1712 = 'missed mark'
  17989 = 'Missing'
  9496 = 'missing marks'
  4567 = 'mm'
  1855 = 'Mode'
  15104 = 'Mode: %s'
  4697 = 'mode=%d'
  7218 = 'Motion'
  1942 = 'MOTION'
  3737 = 'Move Done'
  3074 = 'Move Z axis down after cleaning'
  2526 = 'Moving'
  5512 = 'Moving > Min.Speed for production'
  1914 = 'Name'
  10904 = 'Nbr Marks'
  1164 = 'Nbr Uses'
  13510 = 'No'
  17976 = 'no'
  784 = 'node'
  13171 = 'normal'
  16031 = 'Normal'
  1861 = 'Not all frames contain teach p'
  875 = 'Not all frames contain teach points'
  3138 = 'not engaged (Service)'
  11 = 'Not enough teach points for mode'
  2433 = 'NOTE: might be setup internally'
  10357 = 'num of grid points for job'
  1860 = 'num: %d'
  1919 = 'number exports, max:100'
  4362 = 'number of attached cts'
  385 = 'NumCTs'
  7300 = 'O'
  4393 = 'Off delay'
  5911 = 'OK'
  1847 = 'Open Shutter'
  511 = 'OPERATIONS'
  12010 = 'OtherMarks'
  1406 = 'Out Dir'
  2788 = 'Out Path'
  13228 = 'Outlet'
  5862 = 'OutputPath'
  2864 = 'Outside of machine'
  2527 = 'P\n%s'
  1774 = 'P%d'
  7846 = 'P1'
  18520 = 'P2'
  16371 = 'P3'
  2574 = 'P4'
  3836 = 'p: %d'
  1868 = 'PA'
  1923 = 'pA'
  11770 = 'PA1 WorkerPos'
  709 = 'Park'
  4056 = 'ParkPosition'
  1926 = 'pB'
  4279 = 'Permanent activation'
  1283 = 'PG '
  12785 = 'PG enable'
  3101 = 'PG XPosition'
  3591 = 'PG XPosition [m]'
  6193 = 'PG XPosition [um]'
  500 = 'PG1'
  501 = 'PG2'
  1192 = 'PG: %s'
  3020 = 'Place'
  1169 = 'PM'
  5877 = 'PM Distance to prev PM [m]'
  2049 = 'PM Distance to prev. PM [m]'
  336 = 'PM Distance to previvous PM [m]'
  20630 = 'PM in maintenance position'
  18050 = 'PM in printing position'
  2652 = 'PM Pos mech. to current Master'
  2540 = 'PM Pos mech. to current Master PU'
  9645 = 'PM position'
  2884 = 'PM position on main tracker'
  327 = 'PM position to prev'
  4663 = 'PM position to previous'
  18635 = 'PM X to Master Distance [m]'
  1121 = 'PmPosition=%0.5f   NOTE: PmPosition might be setup/added internally'
  5363 = 'Points'
  8746 = 'Port: %s'
  21704 = 'Pos'
  401 = 'Position'
  3032 = 'Position A'
  3038 = 'Position B'
  3044 = 'Position p1'
  3050 = 'Position p2'
  4232 = 'Position p3'
  4240 = 'Position p4'
  4208 = 'Position [mm]'
  7104 = 'Position [m]'
  8615 = 'Position [SubPx]'
  4770 = 'POSITIONS'
  1116 = 'Pre-StartOffset'
  566 = 'Pre-StartShiftFactor'
  2951 = 'Pre-StartShiftOffset'
  2554 = 'PreStart'
  5281 = 'PreStart (Factor/Offset)'
  7030 = 'PreStart ShiftFactor'
  5299 = 'PreStart ShiftOffset'
  10387 = 'PRG_PRINT'
  164 = 'Print'
  738 = 'Print '
  1180 = 'Print Direction (1=reverse)'
  14325 = 'Print enabled'
  1049 = 'Print Position'
  734 = 'Print Unit'
  4516 = 'Print unit (max %d)'
  12625 = 'Print1'
  3057 = 'Print2'
  5115 = 'Printhead 1'
  3223 = 'Printhead 2'
  8129 = 'PrintModule'
  18556 = 'PrintOffsetX'
  3350 = 'PrintOffsetY'
  10191 = 'PrintON'
  1536 = 'PrintPosition'
  4542 = 'PrintResolution'
  529 = 'PrintSpeed'
  4012 = 'PrintUnit temp at calibration [°C]: %1.1f'
  2680 = 'PrintUnit temperature [°C]: %1.1f'
  2360 = 'processed grid points'
  11146 = 'Produced: %s'
  5301 = 'ProductionSpeed'
  5878 = 'PU'
  4979 = 'PU 4p correction'
  2391 = 'PU 4p correction PLC'
  7392 = 'PU 4p correction PUC'
  6196 = 'PU banana correction'
  18230 = 'Pulse from encoder'
  21913 = 'Pulse Speed'
  8792 = 'Pump set [%]'
  593 = 'Purge'
  721 = 'Purge after Capping'
  13588 = 'PuToWorker'
  4094 = 'PyBusy'
  1213 = 'PyDefDone'
  12566 = 'PyError'
  2980 = 'PyId'
  11014 = 'PyPos'
  11517 = 'Python'
  1054 = 'Python Interface'
  10985 = 'PyUpd'
  90 = 'R'
  1066 = 'r: %d'
  7744 = 'r:%d'
  6096 = 'reached'
  150 = 'Ready'
  703 = 'Ref'
  11729 = 'reference'
  468 = 'Refresh'
  1058 = 'Reg.Points'
  3463 = 'Release from machine'
  1292 = 'Repeat History'
  3912 = 'RepeatLength'
  2586 = 'Reset'
  7014 = 'Reverse'
  4287 = 'Reverse cleaning drive'
  1181 = 'Reverse Direction'
  1955 = 'row'
  13758 = 'Rows: %d'
  4445 = 'Run down delay'
  3142 = 'Running'
  2929 = 'rx'
  10078 = 'RxCtr'
  2932 = 'ry'
  407 = 'S'
  5317 = 's'
  5767 = 's: %d'
  3768 = 'Safe Running Condition'
  3745 = 'Safety'
  17962 = 'Safety cover'
  15672 = 'Safety doors'
  8652 = 'Safety ok'
  3730 = 'SafetyConditionOK'
  3186 = 'Save CT'
  12285 = 'scanned points'
  19355 = 'Scrap:    %s'
  8666 = 'Script alive'
  6352 = 'Sector msg'
  7047 = 'Sel PH : %d '
  6555 = 'Selected for printing'
  14908 = 'Selection MasterModule'
  5838 = 'Send Loop test message'
  3413 = 'Sensor detect errors'
  742 = 'Serv'
  3783 = 'Service'
  2692 = 'ServiceEnabled'
  4356 = 'Set'
  1665 = 'Set value'
  5081 = 'Setpoint #1 [%]'
  2548 = 'Setpoint #2 [%]'
  1673 = 'Setpoint #3 [%]'
  3808 = 'Setpoint #4 [%]'
  2275 = 'Setpoint intensity'
  4255 = 'Setpoint [%]'
  61 = 'Settings'
  14005 = 'Setup'
  1795 = 'Setup new Time'
  308 = 'Setup SpeedCompensation'
  986 = 'Setup [mm]'
  21074 = 'Setup [m]'
  5118 = 'Sh'
  15331 = 'Sheet detect supervision'
  2258 = 'SheetCycle'
  1382 = 'SheetDetect'
  3305 = 'SheetGap'
  2344 = 'SheetGap [mm]'
  1697 = 'SheetLength'
  2532 = 'SheetLength [mm]'
  822 = 'SheetSpeed'
  1118 = 'SheetSpeed [m/min]'
  2238 = 'SheetTrigger'
  5168 = 'ShiftFact'
  6358 = 'ShiftOffs'
  6611 = 'Show Details'
  21803 = 'Show PC'
  20887 = 'Show PH'
  727 = 'Shutter'
  1344 = 'Sim'
  5078 = 'Sim MarkCamera'
  18626 = 'Sim MarkDetection'
  10659 = 'Sim Module'
  5898 = 'Sim position'
  2393 = 'Sim Position %0.3f [m/s]'
  12400 = 'simulate'
  11236 = 'Simulation'
  450 = 'Simulation auto-trigger'
  159 = 'Simulation enable'
  3368 = 'simulation mode'
  19662 = 'Specific Modules'
  2330 = 'Speed'
  6688 = 'speed compensationa active'
  10686 = 'Speed Exceeded'
  15504 = 'Speed m/min'
  181 = 'Speed m/s'
  2930 = 'Speed valid'
  105 = 'Speed [m/min]'
  1484 = 'Speed [m/min] %0.03f [m/s]'
  37 = 'Speed [m/min] %0.03s [m/s]'
  1515 = 'Speed [m/min] %s [m/s]'
  12089 = 'Speed [m/s]'
  1654 = 'Speed [sheet/h]'
  1220 = 'SpeedComp'
  18209 = 'SpeedExeeded'
  3813 = 'SPEEDS'
  12942 = 'sq:%0.3f'
  2356 = 'square length [mm]'
  12697 = 'square length [m]'
  1229 = 'St'
  4781 = 'Standby'
  5000 = 'Start Cleaning'
  20519 = 'start overrun'
  8343 = 'Start overrun'
  508 = 'Start Purge'
  4358 = 'Start up offset'
  9434 = 'start update'
  8070 = 'Started'
  14044 = 'StartMark'
  1620 = 'StartOffs'
  1680 = 'State'
  7664 = 'State name'
  18 = 'Status'
  3715 = 'STATUS'
  12536 = 'Step'
  12315 = 'Stop'
  2267 = 'Stop -> 0 [m/s]'
  17146 = 'Stop Request'
  5135 = 'SubPx'
  9498 = 'Substrate Gap (sim)'
  806 = 'Substrate Length'
  11702 = 'Substrate Width'
  3446 = 'SubstrateLength'
  1519 = 'SubstrateLength effect.'
  687 = 'SystemReady'
  5130 = 't: %d'
  4402 = 'Target'
  9116 = 'Target speed'
  5478 = 'Target speed reached'
  1960 = 'TargetSpeed [m/s]'
  11241 = 'TcpIpClient'
  5655 = 'Teach'
  15269 = 'teached marks'
  19842 = 'Teached Marks: %d'
  2734 = 'teached points'
  21 = 'TeachP'
  460 = 'TeachPoints first frame'
  1422 = 'TeachPoints in first frame'
  10982 = 'Temp at calibration [°C]: %1.1f'
  62 = 'Test'
  4175 = 'TEst'
  2921 = 'Test mode!'
  1251 = 'Test1'
  2109 = 'Test2'
  122 = 'Time'
  8956 = 'To row: %d'
  14553 = 'TODO'
  1520 = 'Tolerance'
  5472 = 'too long'
  3304 = 'too long$'
  8448 = 'Too short'
  3182 = 'too short'
  5716 = 'Total columns'
  7951 = 'tr:%0.3f'
  5292 = 'TrackPos'
  3091 = 'triangle length [mm]'
  16029 = 'triangle length [m]'
  7998 = 'Trigger active'
  228 = 'Trigger Armed'
  2681 = 'TriggerDistance'
  1388 = 'TriggerPulseLength'
  13192 = 'TrigToCam'
  7368 = 'T_PL1'
  1074 = 'T_PL2'
  11769 = 'update done'
  1306 = 'Use Global Grid Shift'
  5046 = 'UseCameraTrigger'
  10877 = 'UseCameraTriggerFeedback'
  5635 = 'UseLength'
  18311 = 'UsePerRepeat'
  3104 = 'v'
  5948 = 'V'
  4271 = 'VACUUM'
  4759 = 'Vacuum pump'
  2945 = 'valid'
  2158 = 'vbn'
  12744 = 'Verbose'
  1735 = 'Verbose mode'
  745 = 'Wait'
  746 = 'Waiting'
  4224 = 'Warning level'
  11338 = 'With Mark'
  3026 = 'Work'
  9075 = 'Worker enable'
  18138 = 'Worker PrintEnable'
  19928 = 'WorkerCamera'
  15457 = 'WorkercCamera'
  13015 = 'WorkerDeform'
  4305 = 'WorkerDeformation'
  11590 = 'WorkerDelete'
  2580 = 'WorkerOffset'
  670 = 'WorkerOffset (PU/PM/PG)'
  1622 = 'WorkerPos (Attach)'
  12 = 'WorkerPos (to Master PM)'
  7284 = 'WorkerPosition'
  13745 = 'WorkerPrint %s'
  8780 = 'WorkerPrint enable'
  2559 = 'WorkerPrint1'
  6462 = 'WorkerPrint1 Line1'
  2497 = 'WorkerPrint2'
  14277 = 'WorkerPrint[1]'
  13424 = 'WorkerPrint[2]'
  6175 = 'WorkerPrint_fPrintStartOffset'
  6394 = 'WorkerPython'
  2890 = 'WorkerVerify'
  3090 = 'Working  pCT'
  2940 = 'x'
  9460 = 'X Ref'
  12401 = 'x [px 4800dpi]'
  886 = 'X0'
  15726 = 'X0 [SubPx]'
  15794 = 'X0: %d'
  4503 = 'x=%0.4f'
  17127 = 'XD: %d'
  887 = 'XS'
  194 = 'XS (+offset + Corrections X)'
  10930 = 'x_P [mm]'
  3312 = 'x_ref'
  14137 = 'x_ref_P [mm]'
  2942 = 'y'
  1070 = 'y [px 4800dpi]'
  8833 = 'Y-Resolution at calibration [dpi]: %1.4f'
  1 = 'y-shift'
  4527 = 'y=%0.4f'
  9660 = 'Yes'
  2488 = 'yes'
  5240 = 'y_max'
  1071 = 'y_P [mm]'
  10734 = 'y_ref'
  7467 = 'y_ref_P [mm]'
  2747 = 'Z Axis'
  1073 = '[%s]'
  13426 = '[-] WebStrech calculated'
  5404 = '[1] CT Id=%d'
  1166 = '[2] CT Id=%d'
  17264 = '[m/s] Max. Speed'
  11491 = '[m/s] Speed'
  3807 = '[mm/C]'
  1135 = '[mm]'
  4403 = '[m]'
  3395 = '[m] HeadGap'
  19619 = '[m] LateralRegister'
  8220 = '[m] Module2ToModule3'
  18328 = '[m] SubstrateLength'
  19359 = '[m] SubstrateThickness'
  2475 = '[p/um] Encoder resolution'
  17520 = '[um] SubstrateThickness'
  3480 = '^'
END_TEXTLIST

// ---- POUs/Machine/ExhaustSystem/_VISU_ExhaustSystemPrint.TcVIS
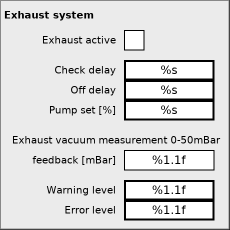
VISUALIZATION _VISU_ExhaustSystemPrint  // 230x230
VAR_IN_OUT
	mInst : FB_ExhaustSystemPrint;
END_VAR
    Rectangle (0,0 230x230)
    Rectangle (1,5 192x20), "Exhaust system"
    Rectangle (29,60 90x20), "Check delay"
    Rectangle (124,60 90x20), "%s", text variable: mInst.tR_VacuumCheckDelay
        OnMouseDown: write the text variable via Edit
    Rectangle (29,80 90x20), "Off delay"
    Rectangle (124,80 90x20), "%s", text variable: mInst.tR_FUOffDelay
        OnMouseDown: write the text variable via Edit
    RoundedRectangle (124,30 20x20), colour toggle: mInst.bO_FUActivate
    Rectangle (19,30 100x20), "Exhaust active"
    Rectangle (9,130 220x20), "Exhaust vacuum measurement 0-50mBar"
    Rectangle (29,150 90x20), "feedback [mBar]"
    Rectangle (124,150 90x20), "%1.1f", text variable: mInst.fL_VacuumAnalogLevelMBar
    Rectangle (29,180 90x20), "Warning level"
    Rectangle (124,180 90x20), "%1.1f", text variable: mInst.fR_VacuumWarningLevelMBar
        OnMouseDown: write the text variable via Edit
    Rectangle (29,200 90x20), "Error level"
    Rectangle (124,200 90x20), "%1.1f", text variable: mInst.fR_VacuumErrorLevelMBar
        OnMouseDown: write the text variable via Edit
    Rectangle (29,100 90x20), "Pump set [%]"
    Rectangle (124,100 90x20), "%s", text variable: mInst.iR_VacuumPumpSetPercent
        OnMouseDown: write the text variable via Edit, min 0, max 100
END_VISUALIZATION

// ---- POUs/Machine/PowerControl/_VISU_PowerControl.TcVIS
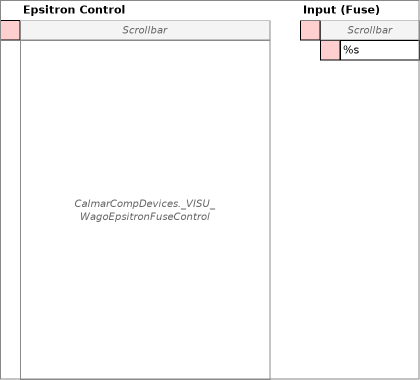
VISUALIZATION _VISU_PowerControl  // 420x380
VAR_IN_OUT
	mInst : FB_PowerControl;
END_VAR
    Frame (20,40 250x340)
        shows CalmarCompDevices._VISU_WagoEpsitronFuseControl(m_Inst_Fb := mInst.pEpsitronsInst[mInst.nEpsitronViewSel]^)
    RoundedRectangle (320,40 20x20), colour toggle: mInst.pFuseInputs[mInst.nFuseViewSel]^
    Scrollbar (320,20 100x20)
        p2245068023: mInst.nFuseInputsRegistered
        p1057716461: mInst.nFuseViewSel
    Rectangle (340,40 80x20), "%s", tooltip "%s", text variable: mInst.aFuseNames[mInst.nFuseViewSel]
        p4168582468: mInst.aFuseNames[mInst.nFuseViewSel]
    RoundedRectangle (300,20 20x20), tooltip "All Inputs ok", colour toggle: mInst.bO_AllFuseOk
    RoundedRectangle (0,20 20x20), tooltip "All Epsitron OK", colour toggle: mInst.bO_AllEpsitronOk
    Scrollbar (20,20 250x20)
        p2245068023: mInst.nEpsitronsRegistered
        p1057716461: mInst.nEpsitronViewSel
    Rectangle (20,0 250x20), "Epsitron Control"
    Rectangle (300,0 120x20), "Input (Fuse)"
END_VISUALIZATION

// ---- POUs/Machine/UV_LED_Modul/_VISU_UvLedModule.TcVIS
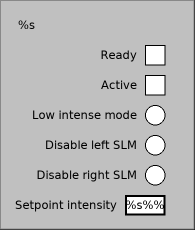
VISUALIZATION _VISU_UvLedModule  // 195x230
VAR_IN_OUT
  m_Inst_Fb   : FB_UvLedModule;
END_VAR
    Rectangle (0,0 195x230), colour variable: m_Inst_Fb._nColorRGB
        p2167032090: m_Inst_Fb._nColorRGB
        p3092690914: 16#FFFF0000
        p3450524324: 16#FF000000
    Rectangle (15,15 155x20), "%s", text variable: m_Inst_Fb._sColorName
    RoundedRectangle (145,45 20x20), colour toggle: m_Inst_Fb.IbReady
    Rectangle (20,45 120x20), "Ready"
    RoundedRectangle (145,75 20x20), colour toggle: m_Inst_Fb._bActivate
    Rectangle (20,75 120x20), "Active"
    Ellipse (145,105 20x20), colour toggle: m_Inst_Fb.RbLowIntenseMode
        toggle m_Inst_Fb.RbLowIntenseMode
    Rectangle (20,105 120x20), "Low intense mode"
    Ellipse (145,135 20x20), colour toggle: m_Inst_Fb.RbDisableLeft
        toggle m_Inst_Fb.RbDisableLeft
    Rectangle (20,135 120x20), "Disable left SLM"
    Ellipse (145,165 20x20), colour toggle: m_Inst_Fb.RbDisableRight
        toggle m_Inst_Fb.RbDisableRight
    Rectangle (20,165 120x20), "Disable right SLM"
    Rectangle (11,195 109x20), "Setpoint intensity"
    Rectangle (125,195 40x20), "%s%%", text variable: m_Inst_Fb.RnIntensitySetpoint
        OnMouseDown: write the text variable via VisuDialogs.Numpad, min m_Inst_Fb.CnMinIntensitySetpoint, max m_Inst_Fb.CnMaxIntensitySetpoint
END_VISUALIZATION

// ---- POUs/Print/Camera/_VISU_CameraBase.TcVIS
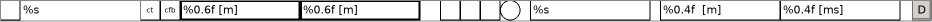
VISUALIZATION _VISU_CameraBase  // 932x22
VAR_IN_OUT
	m_Inst : FB_CameraBase;
END_VAR
    Rectangle (660,0 120x20), "%0.4f [m]", tooltip "TriggerDistance", text variable: m_Inst._fTriggerDistance
        OnMouseDown: write the text variable via Default
    Rectangle (780,0 120x20), "%0.4f [ms]", tooltip "TriggerPulseLength", text variable: m_Inst._fTriggerPulseLength
        OnMouseDown: write the text variable via Default
    RoundedRectangle (440,0 20x20), tooltip "Initialized", colour toggle: m_Inst._bInitialized
    RoundedRectangle (460,0 20x20), tooltip "Camera sink", colour toggle: m_Inst._iCameraSink <> 0
    RoundedRectangle (480,0 20x20), tooltip "Camera trigger", colour toggle: m_Inst._iCameraTrigger <> 0
    Ellipse (500,0 20x20), tooltip "simulate"
        toggle m_Inst._bSimulate
    Frame (0,0 432x22)
        shows _VISU_CameraBaseSetting(m_Inst := m_Inst)
    Button (912,0 20x20), "D", tooltip "Camera Detail: %s", invisible if: m_Inst._sVisuName='unvailable'
        p4168582468: m_Inst._sVisuName
        OnMouseClick: change screen: AssignExpression m_Inst._sVisuName
    Rectangle (530,0 120x20), "%s", tooltip "configured camera mode, active=%s", text variable: m_Inst._eCameraMode
        p4168582468: m_Inst.eCameraMode
        OnMouseDown: write the text variable via Default
END_VISUALIZATION

// ---- POUs/Print/Camera/_VISU_CameraBaseSetting.TcVIS
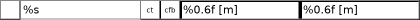
VISUALIZATION _VISU_CameraBaseSetting  // 420x20
VAR_IN_OUT
	m_Inst : FB_CameraBase;
END_VAR
    Rectangle (300,0 120x20), "%0.6f [m]", tooltip "CameraToPrintUnit", text variable: m_Inst._fCameraToPrintOffset
        OnMouseDown: write the text variable via Default
    Rectangle (180,0 120x20), "%0.6f [m]", tooltip "DetectToCamera", text variable: m_Inst._fDetectToCameraOffset
        OnMouseDown: write the text variable via Default
    RoundedRectangle (140,0 20x20), "ct", tooltip "UseCameraTrigger", colour toggle: m_Inst._bUseCameraTrigger
    RoundedRectangle (160,0 20x20), "cfb", tooltip "UseCameraTriggerFeedback", colour toggle: m_Inst._bUseCameraTriggerFeedback
    Rectangle (20,0 120x20), "%s", text variable: m_Inst.sName, colour toggle: m_Inst._bActivated <> 0
    RoundedRectangle (0,0 20x20), tooltip "Camera activated", colour toggle: m_Inst._bActivated <> 0
END_VISUALIZATION

// ---- POUs/Print/Camera/_VISU_CameraTcpIp.TcVIS
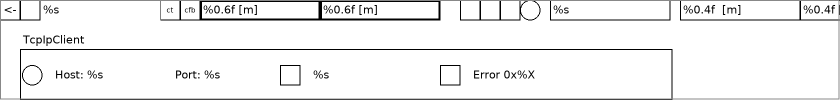
VISUALIZATION _VISU_CameraTcpIp  // 840x100
VAR_IN_OUT
	m_Inst : FB_CameraTcpIp;
END_VAR
    Rectangle (20,49 652x51)
    Frame (20,0 820x23)
        shows _VISU_CameraBase(m_Inst := m_Inst)
    Frame (22,65 240x21)
        shows _VISU_CameraTcpIpSetting(m_Inst := m_Inst)
    RoundedRectangle (0,0 20x20), "<-"
        OnMouseClick: change screen: Previous 
    RoundedRectangle (280,65 20x20), tooltip "Connected", colour toggle: m_Inst._pFbTcpIpClient^.bConnected
    RoundedRectangle (440,65 20x20), tooltip "Error", colour toggle: m_Inst._bConnectionError
    Rectangle (310,65 120x20), "%s", text variable: m_Inst._pFbTcpIpClient^.eStep
    Rectangle (470,65 120x20), "Error 0x%X", text variable: m_Inst._pFbTcpIpClient^.nErrId
    Rectangle (20,30 120x20), "TcpIpClient"
END_VISUALIZATION

// ---- POUs/Print/Camera/_VISU_CameraTcpIpSetting.TcVIS
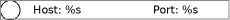
VISUALIZATION _VISU_CameraTcpIpSetting  // 230x20
VAR_IN_OUT
	m_Inst : FB_CameraTcpIp;
END_VAR
    Ellipse (0,0 20x20)
        toggle m_Inst._pFbTcpIpClient^.bEnable
    Rectangle (30,0 120x20), "Host: %s", tooltip "Camera ip address", text variable: m_Inst._pFbTcpIpClient^.sRemoteHost
    Rectangle (150,0 80x20), "Port: %s", tooltip "camera port", text variable: m_Inst._pFbTcpIpClient^.nRemotePort
END_VISUALIZATION

// ---- POUs/Print/Camera/_VISU_CameraTrigger.TcVIS
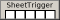
VISUALIZATION _VISU_CameraTrigger  // 60x20
VAR_IN_OUT
	mInst : FB_CameraTrigger;
END_VAR
    RoundedRectangle (0,0 60x20), tooltip "Trigger Armed", colour toggle: mInst.bTriggerArmed
    RoundedRectangle (15,10 10x10), tooltip "Speed valid", colour toggle: mInst.bSpeedValid
    RoundedRectangle (25,10 10x10), tooltip "AutomaticMode or ManualTeach", colour toggle: mInst._bCamManualTeachMode OR mInst.bI_AutomaticMode
    RoundedRectangle (35,10 10x10), tooltip "Inhibit trigger", colour toggle: NOT mInst.bInhibitTrigger
    RoundedRectangle (45,10 10x10), tooltip "HwEnable", colour toggle: mInst.bI_HwEnable
    RoundedRectangle (5,10 10x10), tooltip "Init ok", colour toggle: mInst.bInitOk
    Rectangle (0,0 60x10), "SheetTrigger", tooltip "SheetDetect"
END_VISUALIZATION

// ---- POUs/Print/Camera/_VISU_DeformationPoint.TcVIS
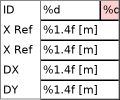
VISUALIZATION _VISU_DeformationPoint  // 120x100
VAR_IN_OUT
	m_Inst : ST_DeformationPointAccurate;
END_VAR
    Rectangle (40,0 60x20), "%d", text variable: m_Inst.index
    Rectangle (0,0 40x20), "ID"
    Rectangle (40,20 80x20), "%1.4f [m]", text variable: m_Inst.x_ref
    Rectangle (0,20 40x20), "X Ref"
    Rectangle (40,40 80x20), "%1.4f [m]", text variable: m_Inst.y_ref
    Rectangle (0,40 40x20), "X Ref"
    Rectangle (40,60 80x20), "%1.4f [m]", text variable: m_Inst.dx
    Rectangle (0,60 40x20), "DX"
    Rectangle (40,80 80x20), "%1.4f [m]", text variable: m_Inst.dy
    Rectangle (0,80 40x20), "DY"
    Rectangle (100,0 20x20), "%d", text variable: m_Inst.valid
END_VISUALIZATION

// ---- POUs/Print/Camera/_VISU_LineCamera.TcVIS
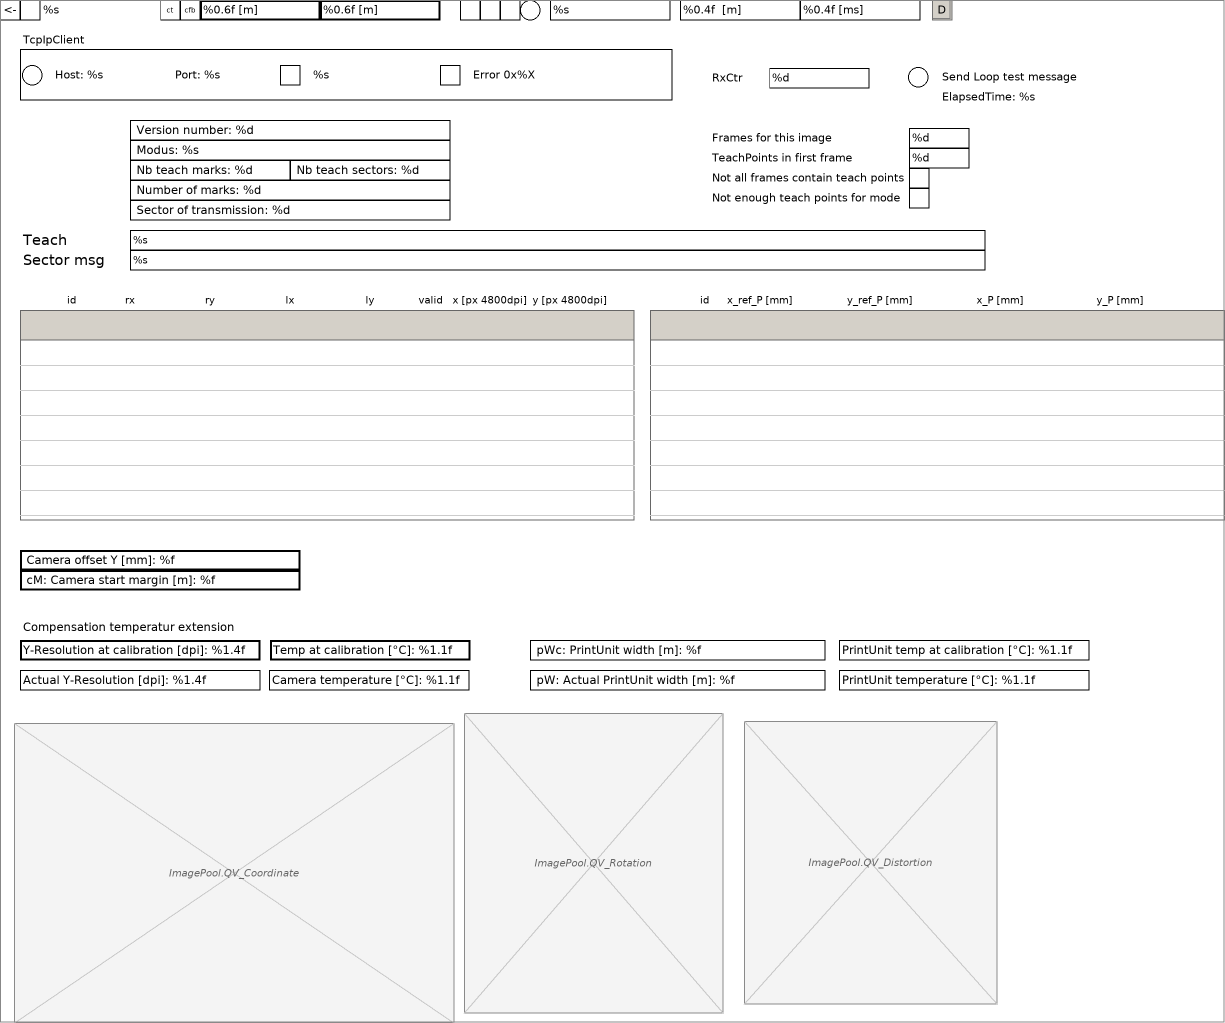
VISUALIZATION _VISU_LineCamera  // 1225x1023
VAR_INPUT
	m_Inst : FB_LineCamera;
END_VAR
    Rectangle (20,230 100x20), "Teach"
    Rectangle (130,230 855x20), "%s", text variable: m_Inst.sTeach
    Rectangle (130,120 320x20), "Version number: %d", text variable: m_Inst.nNbVersion
    Rectangle (130,160 160x20), "Nb teach marks: %d", text variable: m_Inst.nNbMarksTeach
    Table (20,310 614x210), data array: m_Inst.sCameraPoints
        p1128707560: GVL_Camera.cMaxNbMarks
        p2501879983: m_Inst.stCameraResult[INDEX].y_ref_Print
        p7306298: m_Inst.stCameraResult[INDEX].x_teach_Print
        p1933151965: m_Inst.stCameraResult[INDEX].y_teach_Print
        p3863566920: m_Inst.stCameraResult[INDEX].x_Print
        p2192122294: m_Inst.stCameraResult[INDEX].y_Print
        p3854506369: m_Inst.sCameraPoints[INDEX].id
        p1892666644: m_Inst.sCameraPoints[INDEX].x_ref
        p338671338: m_Inst.sCameraPoints[INDEX].y_ref
        p2170511999: m_Inst.sCameraPoints[INDEX].lx
        p3723444502: m_Inst.sCameraPoints[INDEX].ly
        p1218418051: m_Inst.sCameraPoints[INDEX].valid
    Rectangle (90,290 80x20), "rx"
    Rectangle (170,290 80x20), "ry"
    Rectangle (250,290 80x20), "lx"
    Rectangle (330,290 80x20), "ly"
    Rectangle (450,290 80x20), "x [px 4800dpi]"
    Rectangle (530,290 80x20), "y [px 4800dpi]"
    Rectangle (406,290 50x20), "valid"
    Rectangle (130,200 320x20), "Sector of transmission: %d", text variable: m_Inst.nSector
    Rectangle (530,640 295x20), "pWc: PrintUnit width [m]: %f", text variable: m_Inst._fPrintUnitWidthTC
    Image (14,723 440x300), image: ImagePool.QV_Coordinate
    Image (464,713 259x300), image: ImagePool.QV_Rotation
    Image (744,721 253x283), image: ImagePool.QV_Distortion
    Rectangle (20,250 100x20), "Sector msg"
    Rectangle (130,250 855x20), "%s", text variable: m_Inst.sMemLastMessage
    Rectangle (720,290 80x20), "x_ref_P [mm]"
    Rectangle (840,290 80x20), "y_ref_P [mm]"
    Rectangle (960,290 80x20), "x_P [mm]"
    Rectangle (1080,290 80x20), "y_P [mm]"
    Table (650,310 575x210), data array: m_Inst.sTeachPoints
        p1128707560: GVL_Camera.cMaxNbMarks
        p746581629: m_Inst.sTeachPoints[INDEX].y_Print
        p3104783080: m_Inst.stCameraResult[INDEX].x_ref_Print
        p2501879983: m_Inst.stCameraResult[INDEX].y_ref_Print
        p7306298: m_Inst.stCameraResult[INDEX].x_teach_Print
        p1933151965: m_Inst.stCameraResult[INDEX].y_teach_Print
        p3863566920: m_Inst.stCameraResult[INDEX].x_Print
        p2192122294: m_Inst.stCameraResult[INDEX].y_Print
        p3854506369: m_Inst.sTeachPoints[INDEX].id
        p1892666644: m_Inst.sTeachPoints[INDEX].x_ref_Print
        p338671338: m_Inst.sTeachPoints[INDEX].y_ref_Print
        p2170511999: m_Inst.sTeachPoints[INDEX].x_teach_Print
        p3723444502: m_Inst.sTeachPoints[INDEX].y_teach_Print
        p1218418051: m_Inst.sTeachPoints[INDEX].x_Print
    Rectangle (20,640 240x20), "Y-Resolution at calibration [dpi]: %1.4f", text variable: m_Inst.fCameraResolution
        OnMouseDown: write the text variable via Edit
    Rectangle (20,670 240x20), "Actual Y-Resolution [dpi]: %1.4f", text variable: m_Inst.fCameraRealResolution
    Rectangle (269,670 200x20), "Camera temperature [°C]: %1.1f", text variable: m_Inst.fCameraTemp
    Rectangle (270,640 200x20), "Temp at calibration [°C]: %1.1f", text variable: m_Inst.fCameraCalTemp
        OnMouseDown: write the text variable via Edit
    Rectangle (839,640 250x20), "PrintUnit temp at calibration [°C]: %1.1f", text variable: m_Inst._fPrintUnitCalTemp
    Rectangle (839,670 250x20), "PrintUnit temperature [°C]: %1.1f", text variable: m_Inst.fPrintUnitTemp
    Rectangle (20,617 245x20), "Compensation temperatur extension"
    Rectangle (530,670 295x20), "pW: Actual PrintUnit width [m]: %f", text variable: m_Inst.fPrintUnitWidthTAct
    Rectangle (130,180 320x20), "Number of marks: %d", text variable: m_Inst.nNbMarks
    Rectangle (20,550 280x20), "Camera offset Y [mm]: %f", text variable: m_Inst.fCameraAdjustmentY
        OnMouseDown: write the text variable via Edit
    Rectangle (20,570 280x20), "cM: Camera start margin [m]: %f", text variable: m_Inst.fCameraStartMargin
        OnMouseDown: write the text variable via Edit
    Rectangle (130,140 320x20), "Modus: %s", text variable: m_Inst.sModus
    Frame (0,0 861x79)
        shows _VISU_CameraTcpIp(m_Inst := m_Inst)
    Rectangle (290,160 160x20), "Nb teach sectors: %d", text variable: m_Inst.nNbSectorTeach
    Ellipse (908,67 20x20)
        tap m_Inst._bTestTx
    Rectangle (769,68 100x20), "%d", text variable: m_Inst.nRxMsg
    Rectangle (709,68 60x20), "RxCtr"
    Rectangle (939,67 161x20), "Send Loop test message"
    Rectangle (939,87 161x20), "ElapsedTime: %s", text variable: m_Inst._sTimeElapsed
    Rectangle (709,128 200x20), "Frames for this image"
    Rectangle (909,128 60x20), "%d", text variable: m_Inst.nNumFrames
    Rectangle (709,148 200x20), "TeachPoints in first frame"
    Rectangle (909,148 60x20), "%d", text variable: m_Inst.nNumPointsPerSectorT[1]
    Rectangle (709,168 200x20), "Not all frames contain teach points"
    RoundedRectangle (909,168 20x20), colour toggle: m_Inst.bNotAllFramesContainTeachPoints
    Rectangle (709,188 200x20), "Not enough teach points for mode"
    RoundedRectangle (909,188 20x20), colour toggle: m_Inst.bNotEnoughTeachPoints
    Rectangle (32,290 80x20), "id"
    Rectangle (690,290 30x20), "id"
END_VISUALIZATION

// ---- POUs/Print/Camera/_VISU_SystronCamera.TcVIS
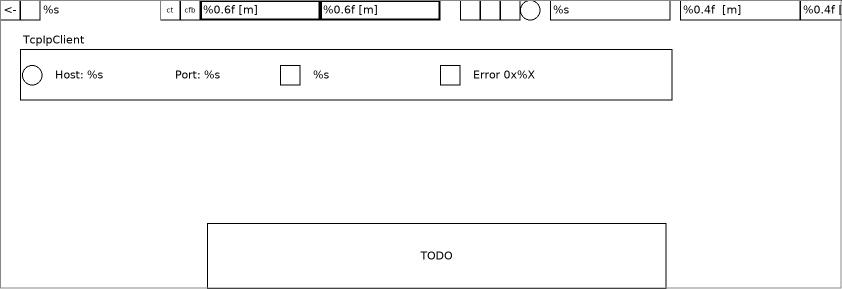
VISUALIZATION _VISU_SystronCamera  // 842x289
    Rectangle (207,223 459x66), "TODO"
    Frame (0,0 842x135)
        shows _VISU_CameraTcpIp(m_Inst := PRG_PRINT.fbLineCamera)
END_VISUALIZATION

// ---- POUs/Print/DefGrid/_Test/Txt_GridTypeSelection.TcTLO
TEXTLIST Txt_GridTypeSelection
  0 = 'Default (dy from StartMark)'
  1 = 'None: Grid calculated dx/dy=0'
  2 = 'Test_AllDxFactor'
  3 = 'Test_AllDyFactor'
  4 = 'Test_DxColFactor'
  5 = 'Test_DyColFactro'
  6 = 'Test_Dx_FirstRowOnlyFactor'
   = ''
END_TEXTLIST

// ---- POUs/Print/DefGrid/_VISU_Templates/E_DeformationType.TcTLO
TEXTLIST E_DeformationType
  0 = 'NoDeformation'
  1 = 'ScriptGrid'
  2 = 'ScriptGridTrend'
  3 = 'LocalMarks1D'
   = ''
END_TEXTLIST

// ---- POUs/Print/DefGrid/_VISU_Templates/_VISU_ContainerDefGrid.TcVIS
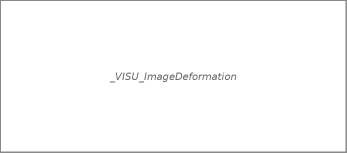
VISUALIZATION _VISU_ContainerDefGrid  // 347x153
VAR_IN_OUT
	m_Inst : FB_ContainerDefGrid;
END_VAR
    Frame (0,0 347x153)
        shows _VISU_ImageDeformation(m_Inst := m_Inst.fBImageDeformation)
END_VISUALIZATION

